C01815=1063.991,309.897,-98.913,173.800,33.597,156.214
C01816=1063.997,310.145,-98.945,173.803,33.601,156.215
C01817=1064.004,310.393,-98.978,173.806,33.605,156.216
C01818=1064.011,310.640,-99.011,173.809,33.609,156.217
C01819=1064.017,310.888,-99.044,173.812,33.614,156.218
C01820=1064.023,311.136,-99.077,173.815,33.618,156.219
C01821=1064.029,311.383,-99.109,173.818,33.622,156.220
C01822=1064.036,311.631,-99.142,173.821,33.626,156.220
C01823=1064.042,311.880,-99.175,173.824,33.631,156.221
C01824=1064.049,312.127,-99.207,173.828,33.635,156.222
C01825=1064.056,312.375,-99.239,173.832,33.640,156.223
C01826=1064.062,312.622,-99.272,173.835,33.644,156.224
C01827=1064.068,312.870,-99.305,173.838,33.648,156.225
C01828=1064.075,313.118,-99.338,173.841,33.652,156.225
C01829=1064.081,313.366,-99.371,173.844,33.657,156.226
C01830=1064.088,313.613,-99.404,173.847,33.661,156.227
C01831=1064.094,313.861,-99.436,173.850,33.665,156.228
C01832=1064.101,314.109,-99.469,173.853,33.670,156.229
C01833=1064.107,314.356,-99.503,173.858,33.674,156.230
C01834=1064.113,314.604,-99.536,173.861,33.679,156.231
C01835=1064.119,314.852,-99.570,173.864,33.683,156.232
C01836=1064.125,315.100,-99.602,173.867,33.688,156.233
C01837=1064.131,315.347,-99.635,173.870,33.692,156.233
C01838=1064.138,315.595,-99.669,173.873,33.697,156.234
C01839=1064.144,315.843,-99.702,173.876,33.701,156.235
C01840=1064.149,316.091,-99.736,173.879,33.705,156.236
C01841=1064.156,316.338,-99.768,173.883,33.710,156.237
C01842=1064.162,316.586,-99.802,173.887,33.714,156.238
C01843=1064.168,316.833,-99.835,173.890,33.719,156.239
C01844=1064.174,317.082,-99.869,173.893,33.723,156.240
C01845=1064.181,317.319,-99.901,173.896,33.728,156.241
C01846=1064.187,317.558,-99.933,173.899,33.732,156.242
C01847=1064.193,317.796,-99.965,173.902,33.736,156.242
C01848=1064.199,318.035,-99.997,173.905,33.741,156.243
C01849=1064.204,318.273,-100.029,173.909,33.745,156.244
C01850=1064.211,318.511,-100.061,173.912,33.749,156.245
C01851=1064.216,318.750,-100.093,173.915,33.754,156.246
C01852=1064.223,318.989,-100.126,173.918,33.758,156.247
C01853=1064.229,319.236,-100.160,173.921,33.762,156.248
C01854=1064.235,319.484,-100.192,173.925,33.767,156.249
C01855=1064.241,319.731,-100.227,173.928,33.772,156.249
C01856=1064.248,319.980,-100.260,173.931,33.776,156.250
C01857=1064.254,320.227,-100.294,173.935,33.781,156.251
C01858=1064.261,320.475,-100.327,173.938,33.785,156.252
C01859=1064.266,320.722,-100.361,173.941,33.789,156.253
C01860=1064.273,320.969,-100.394,173.945,33.794,156.254
C01861=1064.279,321.218,-100.428,173.948,33.799,156.255
C01862=1064.286,321.465,-100.461,173.951,33.803,156.256
C01863=1064.291,321.713,-100.495,173.954,33.808,156.257
C01864=1064.298,321.961,-100.529,173.959,33.813,156.258
C01865=1064.304,322.208,-100.563,173.962,33.817,156.259
C01866=1064.311,322.456,-100.596,173.965,33.821,156.260
C01867=1064.317,322.703,-100.630,173.968,33.826,156.260
C01868=1064.324,322.951,-100.664,173.971,33.831,156.261
C01869=1064.330,323.198,-100.698,173.975,33.835,156.262
C01870=1064.336,323.447,-100.731,173.979,33.840,156.263
C01871=1064.343,323.694,-100.765,173.982,33.844,156.264
C01872=1064.349,323.941,-100.799,173.985,33.849,156.265
C01873=1064.355,324.189,-100.833,173.989,33.853,156.266
C01874=1064.362,324.437,-100.866,173.992,33.858,156.267
C01875=1064.368,324.685,-100.901,173.995,33.863,156.268
C01876=1064.375,324.932,-100.934,173.998,33.867,156.269
C01877=1064.381,325.180,-100.968,174.003,33.872,156.270
C01878=1064.388,325.427,-101.002,174.006,33.876,156.271
C01879=1064.394,325.675,-101.036,174.009,33.881,156.272
C01880=1064.401,325.923,-101.071,174.012,33.886,156.273
C01881=1064.407,326.170,-101.104,174.016,33.890,156.273
C01882=1064.413,326.418,-101.138,174.019,33.895,156.274
C01883=1064.421,326.666,-101.172,174.023,33.899,156.275
C01884=1064.426,326.913,-101.206,174.027,33.904,156.276
C01885=1064.433,327.161,-101.240,174.030,33.909,156.277
C01886=1064.439,327.408,-101.274,174.033,33.913,156.278
C01887=1064.446,327.656,-101.308,174.036,33.918,156.279
C01888=1064.453,327.904,-101.343,174.040,33.923,156.280
C01889=1064.459,328.150,-101.377,174.044,33.928,156.281
C01890=1064.466,328.398,-101.411,174.047,33.932,156.282
C01891=1064.473,328.646,-101.445,174.051,33.936,156.283
C01892=1064.479,328.893,-101.479,174.054,33.941,156.284
C01893=1064.485,329.141,-101.513,174.057,33.946,156.285
C01894=1064.493,329.389,-101.547,174.061,33.950,156.286
C01895=1064.498,329.636,-101.581,174.065,33.955,156.287
C01896=1064.505,329.884,-101.616,174.068,33.960,156.288
C01897=1064.512,330.131,-101.650,174.072,33.965,156.289
C01898=1064.519,330.379,-101.685,174.075,33.969,156.290
C01899=1064.525,330.627,-101.719,174.078,33.974,156.291
C01900=1064.531,330.875,-101.753,174.083,33.979,156.291
C01901=1064.538,331.110,-101.786,174.086,33.983,156.292
C01902=1064.543,331.346,-101.819,174.089,33.987,156.293
C01903=1064.550,331.581,-101.852,174.092,33.992,156.294
C01904=1064.557,331.817,-101.885,174.096,33.997,156.295
C01905=1064.562,332.052,-101.918,174.099,34.002,156.296
C01906=1064.568,332.287,-101.950,174.103,34.006,156.297
C01907=1064.574,332.523,-101.984,174.106,34.010,156.298
C01908=1064.580,332.759,-102.016,174.109,34.015,156.299
C01909=1064.587,333.006,-102.051,174.113,34.020,156.300
C01910=1064.593,333.254,-102.085,174.116,34.025,156.301
C01911=1064.600,333.501,-102.120,174.120,34.030,156.302
C01912=1064.606,333.749,-102.155,174.124,34.034,156.303
C01913=1064.613,333.996,-102.190,174.127,34.040,156.304
C01914=1064.619,334.244,-102.224,174.131,34.044,156.305
C01915=1064.626,334.491,-102.259,174.134,34.049,156.306
C01916=1064.631,334.739,-102.294,174.138,34.054,156.307
C01917=1064.638,334.987,-102.329,174.142,34.059,156.308
C01918=1064.645,335.234,-102.364,174.145,34.064,156.309
C01919=1064.651,335.482,-102.399,174.149,34.068,156.310
C01920=1064.657,335.729,-102.434,174.152,34.073,156.311
C01921=1064.664,335.977,-102.468,174.156,34.078,156.312
C01922=1064.671,336.224,-102.503,174.160,34.083,156.313
C01923=1064.677,336.471,-102.538,174.163,34.088,156.314
C01924=1064.684,336.719,-102.573,174.167,34.093,156.315
C01925=1064.691,336.967,-102.608,174.170,34.098,156.316
C01926=1064.697,337.214,-102.643,174.174,34.103,156.317
C01927=1064.704,337.462,-102.679,174.178,34.107,156.318
C01928=1064.710,337.708,-102.714,174.181,34.113,156.319
C01929=1064.716,337.956,-102.749,174.185,34.118,156.320
C01930=1064.723,338.204,-102.783,174.189,34.122,156.321
C01931=1064.729,338.451,-102.819,174.193,34.128,156.322
C01932=1064.736,338.699,-102.854,174.196,34.132,156.323
C01933=1064.742,338.946,-102.889,174.200,34.138,156.324
C01934=1064.748,339.194,-102.925,174.203,34.142,156.325
C01935=1064.755,339.441,-102.960,174.207,34.147,156.326
C01936=1064.762,339.688,-102.995,174.211,34.153,156.327
C01937=1064.767,339.935,-103.030,174.214,34.157,156.328
C01938=1064.774,340.183,-103.066,174.218,34.163,156.330
C01939=1064.781,340.430,-103.101,174.222,34.168,156.331
C01940=1064.788,340.678,-103.136,174.226,34.172,156.332
C01941=1064.794,340.925,-103.172,174.229,34.178,156.333
C01942=1064.801,341.173,-103.207,174.233,34.183,156.334
C01943=1064.807,341.420,-103.242,174.237,34.188,156.335
C01944=1064.813,341.668,-103.278,174.241,34.193,156.336
C01945=1064.820,341.915,-103.313,174.244,34.198,156.337
C01946=1064.826,342.162,-103.349,174.248,34.203,156.338
C01947=1064.833,342.409,-103.384,174.252,34.208,156.339
C01948=1064.840,342.657,-103.419,174.256,34.213,156.340
C01949=1064.847,342.905,-103.456,174.259,34.218,156.341
C01950=1064.853,343.153,-103.491,174.263,34.223,156.342
C01951=1064.860,343.399,-103.527,174.267,34.228,156.343
C01952=1064.867,343.647,-103.562,174.271,34.233,156.344
C01953=1064.873,343.894,-103.597,174.274,34.239,156.345
C01954=1064.879,344.142,-103.633,174.278,34.244,156.347
C01955=1064.886,344.389,-103.669,174.282,34.249,156.348
C01956=1064.892,344.636,-103.705,174.286,34.254,156.349
C01957=1064.899,344.869,-103.739,174.289,34.259,156.350
C01958=1064.905,345.102,-103.772,174.293,34.264,156.351
C01959=1064.911,345.336,-103.806,174.297,34.269,156.352
C01960=1064.917,345.569,-103.839,174.300,34.274,156.353
C01961=1064.923,345.802,-103.874,174.304,34.279,156.354
C01962=1064.929,346.035,-103.908,174.307,34.284,156.355
C01963=1064.936,346.268,-103.942,174.311,34.288,156.356
C01964=1064.942,346.501,-103.975,174.315,34.294,156.357
C01965=1064.948,346.748,-104.011,174.318,34.299,156.358
C01966=1064.955,346.997,-104.047,174.322,34.304,156.359
C01967=1064.962,347.244,-104.083,174.327,34.309,156.360
C01968=1064.968,347.491,-104.119,174.330,34.314,156.361
C01969=1064.975,347.738,-104.155,174.334,34.320,156.363
C01970=1064.981,347.985,-104.191,174.338,34.325,156.364
C01971=1064.988,348.232,-104.227,174.342,34.331,156.365
C01972=1064.995,348.480,-104.263,174.346,34.336,156.366
C01973=1065.001,348.727,-104.299,174.349,34.341,156.367
C01974=1065.008,348.974,-104.336,174.354,34.346,156.368
C01975=1065.014,349.222,-104.371,174.357,34.351,156.369
C01976=1065.021,349.469,-104.408,174.361,34.357,156.370
C01977=1065.028,349.717,-104.444,174.366,34.362,156.372
C01978=1065.034,349.964,-104.481,174.369,34.367,156.373
C01979=1065.041,350.211,-104.516,174.373,34.373,156.374
C01980=1065.048,350.459,-104.553,174.376,34.378,156.375
C01981=1065.054,350.706,-104.589,174.381,34.384,156.376
C01982=1065.061,350.952,-104.625,174.385,34.389,156.377
C01983=1065.068,351.200,-104.662,174.388,34.394,156.378
C01984=1065.074,351.447,-104.698,174.393,34.400,156.380
C01985=1065.081,351.694,-104.735,174.397,34.405,156.381
C01986=1065.088,351.942,-104.771,174.400,34.411,156.382
C01987=1065.095,352.189,-104.807,174.405,34.416,156.383
C01988=1065.101,352.436,-104.844,174.409,34.422,156.384
C01989=1065.107,352.683,-104.880,174.412,34.427,156.385
C01990=1065.114,352.931,-104.917,174.417,34.432,156.387
C01991=1065.121,353.178,-104.953,174.421,34.438,156.388
C01992=1065.128,353.426,-104.990,174.424,34.443,156.389
C01993=1065.134,353.673,-105.027,174.428,34.449,156.390
C01994=1065.140,353.920,-105.063,174.433,34.454,156.391
C01995=1065.147,354.167,-105.100,174.436,34.460,156.392
C01996=1065.154,354.414,-105.137,174.440,34.466,156.394
C01997=1065.160,354.661,-105.174,174.445,34.471,156.395
C01998=1065.167,354.909,-105.210,174.449,34.477,156.396
C01999=1065.173,355.156,-105.247,174.452,34.482,156.397
C02000=1065.180,355.403,-105.284,174.457,34.488,156.398
C02001=1065.187,355.650,-105.321,174.461,34.493,156.400
C02002=1065.194,355.898,-105.358,174.464,34.499,156.401
C02003=1065.200,356.145,-105.394,174.469,34.505,156.402
C02004=1065.207,356.391,-105.431,174.473,34.510,156.403
C02005=1065.214,356.639,-105.468,174.477,34.516,156.404
C02006=1065.220,356.886,-105.504,174.481,34.521,156.406
C02007=1065.227,357.133,-105.542,174.485,34.527,156.407
C02008=1065.234,357.380,-105.578,174.490,34.533,156.408
C02009=1065.241,357.627,-105.616,174.494,34.538,156.409
C02010=1065.248,357.875,-105.653,174.497,34.544,156.410
C02011=1065.255,358.121,-105.690,174.502,34.549,156.412
C02012=1065.262,358.369,-105.727,174.506,34.555,156.413
C02013=1065.268,358.604,-105.762,174.509,34.561,156.414
C02014=1065.274,358.839,-105.798,174.514,34.566,156.415
C02015=1065.280,359.074,-105.833,174.518,34.572,156.416
C02016=1065.287,359.309,-105.868,174.521,34.577,156.418
C02017=1065.293,359.544,-105.904,174.526,34.582,156.419
C02018=1065.300,359.780,-105.939,174.529,34.588,156.420
C02019=1065.306,360.015,-105.974,174.533,34.593,156.421
C02020=1065.312,360.250,-106.010,174.538,34.599,156.422
C02021=1065.319,360.497,-106.048,174.541,34.605,156.424
C02022=1065.326,360.744,-106.085,174.546,34.610,156.425
C02023=1065.333,360.991,-106.122,174.550,34.616,156.426
C02024=1065.340,361.239,-106.160,174.554,34.622,156.427
C02025=1065.346,361.485,-106.197,174.559,34.628,156.429
C02026=1065.353,361.732,-106.234,174.563,34.634,156.430
C02027=1065.360,361.980,-106.271,174.566,34.639,156.431
C02028=1065.367,362.227,-106.308,174.571,34.645,156.432
C02029=1065.374,362.474,-106.347,174.575,34.651,156.434
C02030=1065.381,362.721,-106.384,174.580,34.657,156.435
C02031=1065.387,362.968,-106.421,174.584,34.663,156.436
C02032=1065.394,363.215,-106.459,174.588,34.669,156.438
C02033=1065.401,363.462,-106.497,174.592,34.675,156.439
C02034=1065.408,363.709,-106.534,174.596,34.680,156.440
C02035=1065.414,363.956,-106.572,174.601,34.687,156.442
C02036=1065.422,364.203,-106.610,174.605,34.692,156.443
C02037=1065.429,364.450,-106.647,174.609,34.698,156.444
C02038=1065.435,364.697,-106.685,174.614,34.704,156.445
C02039=1065.442,364.944,-106.722,174.618,34.710,156.447
C02040=1065.448,365.192,-106.761,174.623,34.717,156.448
C02041=1065.455,365.438,-106.798,174.626,34.722,156.449
C02042=1065.462,365.685,-106.837,174.631,34.728,156.451
C02043=1065.468,365.932,-106.875,174.635,34.735,156.452
C02044=1065.476,366.180,-106.912,174.639,34.740,156.453
C02045=1065.482,366.426,-106.951,174.644,34.747,156.455
C02046=1065.489,366.673,-106.988,174.648,34.753,156.456
C02047=1065.496,366.920,-107.026,174.653,34.759,156.457
C02048=1065.503,367.167,-107.065,174.657,34.765,156.459
C02049=1065.510,367.414,-107.103,174.662,34.771,156.460
C02050=1065.517,367.661,-107.140,174.666,34.777,156.461
C02051=1065.523,367.907,-107.179,174.669,34.783,156.463
C02052=1065.530,368.155,-107.217,174.674,34.790,156.464
C02053=1065.537,368.401,-107.255,174.678,34.796,156.466
C02054=1065.544,368.649,-107.293,174.683,34.802,156.467
C02055=1065.551,368.896,-107.331,174.687,34.808,156.468
C02056=1065.558,369.143,-107.370,174.692,34.814,156.470
C02057=1065.565,369.390,-107.408,174.696,34.820,156.471
C02058=1065.572,369.637,-107.446,174.701,34.826,156.472
C02059=1065.579,369.884,-107.485,174.705,34.832,156.474
C02060=1065.585,370.130,-107.522,174.710,34.839,156.475
C02061=1065.592,370.377,-107.561,174.714,34.845,156.477
C02062=1065.599,370.624,-107.600,174.719,34.852,156.478
C02063=1065.606,370.871,-107.637,174.723,34.858,156.479
C02064=1065.613,371.118,-107.676,174.728,34.864,156.481
C02065=1065.620,371.365,-107.715,174.732,34.870,156.482
C02066=1065.627,371.612,-107.752,174.736,34.876,156.483
C02067=1065.634,371.858,-107.791,174.741,34.883,156.485
C02068=1065.641,372.105,-107.830,174.745,34.889,156.486
C02069=1065.648,372.349,-107.868,174.750,34.896,156.488
C02070=1065.655,372.594,-107.906,174.754,34.902,156.489
C02071=1065.662,372.837,-107.944,174.759,34.908,156.490
C02072=1065.668,373.081,-107.982,174.763,34.914,156.492
C02073=1065.675,373.325,-108.021,174.768,34.921,156.493
C02074=1065.683,373.569,-108.059,174.772,34.927,156.495
C02075=1065.689,373.812,-108.097,174.777,34.933,156.496
C02076=1065.696,374.057,-108.135,174.781,34.940,156.498
C02077=1065.703,374.304,-108.174,174.786,34.946,156.499
C02078=1065.709,374.550,-108.213,174.790,34.953,156.501
C02079=1065.716,374.797,-108.252,174.795,34.960,156.502
C02080=1065.723,375.044,-108.291,174.800,34.966,156.503
C02081=1065.730,375.291,-108.330,174.804,34.972,156.505
C02082=1065.738,375.538,-108.370,174.809,34.979,156.506
C02083=1065.744,375.785,-108.408,174.813,34.985,156.508
C02084=1065.751,376.031,-108.447,174.818,34.992,156.509
C02085=1065.758,376.278,-108.486,174.823,34.999,156.511
C02086=1065.766,376.525,-108.524,174.828,35.006,156.512
C02087=1065.773,376.771,-108.564,174.832,35.012,156.514
C02088=1065.780,377.018,-108.603,174.837,35.018,156.515
C02089=1065.787,377.265,-108.642,174.841,35.025,156.517
C02090=1065.794,377.511,-108.681,174.846,35.032,156.518
C02091=1065.801,377.758,-108.720,174.851,35.039,156.520
C02092=1065.808,378.005,-108.759,174.855,35.045,156.521
C02093=1065.815,378.252,-108.799,174.861,35.052,156.523
C02094=1065.822,378.499,-108.838,174.865,35.059,156.524
C02095=1065.829,378.745,-108.877,174.870,35.065,156.526
C02096=1065.836,378.992,-108.916,174.874,35.072,156.527
C02097=1065.843,379.239,-108.957,174.879,35.079,156.529
C02098=1065.850,379.486,-108.996,174.884,35.085,156.530
C02099=1065.857,379.732,-109.035,174.889,35.092,156.532
C02100=1065.864,379.980,-109.074,174.894,35.099,156.533
C02101=1065.872,380.226,-109.114,174.898,35.106,156.535
C02102=1065.878,380.473,-109.153,174.903,35.113,156.537
C02103=1065.886,380.720,-109.193,174.907,35.119,156.538
C02104=1065.893,380.966,-109.232,174.912,35.126,156.540
C02105=1065.900,381.213,-109.271,174.918,35.133,156.541
C02106=1065.908,381.460,-109.311,174.922,35.140,156.543
C02107=1065.914,381.706,-109.351,174.927,35.147,156.544
C02108=1065.921,381.952,-109.391,174.932,35.154,156.546
C02109=1065.929,382.199,-109.431,174.936,35.161,156.548
C02110=1065.935,382.446,-109.470,174.942,35.168,156.549
C02111=1065.943,382.693,-109.510,174.946,35.175,156.551
C02112=1065.950,382.939,-109.550,174.951,35.182,156.552
C02113=1065.956,383.186,-109.590,174.956,35.189,156.554
C02114=1065.964,383.433,-109.630,174.961,35.196,156.556
C02115=1065.971,383.679,-109.669,174.966,35.203,156.557
C02116=1065.978,383.926,-109.710,174.971,35.210,156.559
C02117=1065.985,384.172,-109.749,174.975,35.217,156.560
C02118=1065.992,384.419,-109.789,174.981,35.224,156.562
C02119=1065.999,384.666,-109.829,174.986,35.232,156.564
C02120=1066.006,384.912,-109.869,174.990,35.238,156.565
C02121=1066.014,385.159,-109.910,174.996,35.246,156.567
C02122=1066.021,385.405,-109.950,175.001,35.253,156.569
C02123=1066.029,385.652,-109.990,175.005,35.260,156.570
C02124=1066.036,385.899,-110.030,175.010,35.267,156.572
C02125=1066.044,386.170,-110.074,175.016,35.275,156.574
C02126=1066.052,386.441,-110.119,175.021,35.283,156.576
C02127=1066.060,386.712,-110.163,175.027,35.291,156.577
C02128=1066.067,386.984,-110.206,175.032,35.299,156.579
C02129=1066.075,387.231,-110.248,175.038,35.306,156.581
C02130=1066.082,387.477,-110.287,175.042,35.314,156.583
C02131=1066.090,387.723,-110.328,175.048,35.321,156.584
C02132=1066.097,387.970,-110.368,175.053,35.328,156.586
C02133=1066.104,388.217,-110.408,175.057,35.336,156.588
C02134=1066.111,388.463,-110.449,175.063,35.343,156.589
C02135=1066.119,388.710,-110.489,175.068,35.350,156.591
C02136=1066.126,388.956,-110.530,175.073,35.358,156.593
C02137=1066.133,389.203,-110.570,175.078,35.365,156.595
C02138=1066.141,389.449,-110.611,175.083,35.372,156.596
C02139=1066.148,389.695,-110.651,175.089,35.380,156.598
C02140=1066.155,389.942,-110.692,175.094,35.387,156.600
C02141=1066.163,390.189,-110.732,175.098,35.395,156.601
C02142=1066.170,390.435,-110.774,175.104,35.402,156.603
C02143=1066.178,390.682,-110.814,175.109,35.410,156.605
C02144=1066.185,390.928,-110.854,175.115,35.417,156.607
C02145=1066.192,391.175,-110.896,175.119,35.425,156.608
C02146=1066.200,391.421,-110.936,175.125,35.432,156.610
C02147=1066.207,391.668,-110.977,175.130,35.440,156.612
C02148=1066.214,391.914,-111.018,175.136,35.448,156.614
C02149=1066.222,392.160,-111.058,175.140,35.455,156.616
C02150=1066.229,392.407,-111.099,175.146,35.463,156.617
C02151=1066.236,392.653,-111.141,175.151,35.471,156.619
C02152=1066.244,392.900,-111.182,175.156,35.478,156.621
C02153=1066.252,393.146,-111.223,175.162,35.486,156.623
C02154=1066.258,393.392,-111.263,175.166,35.494,156.625
C02155=1066.266,393.639,-111.305,175.172,35.501,156.626
C02156=1066.273,393.885,-111.346,175.177,35.509,156.628
C02157=1066.280,394.132,-111.387,175.183,35.517,156.630
C02158=1066.288,394.378,-111.428,175.188,35.525,156.632
C02159=1066.296,394.624,-111.470,175.193,35.533,156.634
C02160=1066.303,394.871,-111.511,175.199,35.541,156.636
C02161=1066.310,395.117,-111.552,175.204,35.548,156.637
C02162=1066.318,395.364,-111.593,175.210,35.556,156.639
C02163=1066.325,395.610,-111.635,175.215,35.564,156.641
C02164=1066.332,395.857,-111.677,175.221,35.572,156.643
C02165=1066.340,396.103,-111.718,175.226,35.580,156.645
C02166=1066.347,396.349,-111.760,175.231,35.588,156.647
C02167=1066.355,396.596,-111.801,175.236,35.596,156.649
C02168=1066.362,396.842,-111.842,175.242,35.604,156.651
C02169=1066.370,397.088,-111.884,175.248,35.612,156.652
C02170=1066.377,397.335,-111.925,175.253,35.620,156.654
C02171=1066.385,397.581,-111.967,175.259,35.628,156.656
C02172=1066.392,397.827,-112.008,175.264,35.636,156.658
C02173=1066.400,398.074,-112.051,175.270,35.645,156.660
C02174=1066.407,398.321,-112.092,175.276,35.653,156.662
C02175=1066.415,398.567,-112.134,175.280,35.661,156.664
C02176=1066.422,398.813,-112.176,175.286,35.669,156.666
C02177=1066.430,399.059,-112.217,175.291,35.677,156.668
C02178=1066.437,399.305,-112.259,175.297,35.685,156.670
C02179=1066.445,399.551,-112.301,175.303,35.694,156.672
C02180=1066.452,399.798,-112.344,175.308,35.702,156.674
C02181=1066.462,400.119,-112.398,175.315,35.713,156.676
C02182=1066.472,400.440,-112.453,175.324,35.724,156.679
C02183=1066.482,400.761,-112.507,175.331,35.734,156.681
C02184=1066.492,401.081,-112.562,175.338,35.745,156.684
C02185=1066.499,401.327,-112.604,175.343,35.754,156.686
C02186=1066.507,401.574,-112.647,175.349,35.762,156.688
C02187=1066.515,401.820,-112.689,175.355,35.771,156.690
C02188=1066.522,402.067,-112.731,175.361,35.779,156.692
C02189=1066.530,402.313,-112.773,175.366,35.788,156.694
C02190=1066.538,402.559,-112.815,175.372,35.796,156.696
C02191=1066.546,402.806,-112.858,175.378,35.804,156.698
C02192=1066.553,403.052,-112.900,175.384,35.813,156.700
C02193=1066.560,403.298,-112.942,175.389,35.822,156.702
C02194=1066.569,403.544,-112.985,175.395,35.830,156.705
C02195=1066.576,403.790,-113.028,175.401,35.839,156.707
C02196=1066.584,404.037,-113.070,175.407,35.848,156.709
C02197=1066.591,404.283,-113.113,175.413,35.856,156.711
C02198=1066.599,404.529,-113.156,175.418,35.865,156.713
C02199=1066.607,404.775,-113.197,175.424,35.874,156.715
C02200=1066.615,405.022,-113.241,175.430,35.882,156.717
C02201=1066.622,405.268,-113.283,175.436,35.891,156.719
C02202=1066.630,405.515,-113.326,175.442,35.900,156.721
C02203=1066.638,405.760,-113.369,175.449,35.909,156.723
C02204=1066.645,406.007,-113.412,175.454,35.917,156.726
C02205=1066.652,406.236,-113.452,175.460,35.926,156.728
C02206=1066.660,406.466,-113.492,175.465,35.934,156.730
C02207=1066.667,406.695,-113.532,175.471,35.942,156.732
C02208=1066.674,406.924,-113.572,175.477,35.951,156.734
C02209=1066.681,407.155,-113.612,175.482,35.959,156.736
C02210=1066.688,407.384,-113.652,175.488,35.968,156.738
C02211=1066.696,407.614,-113.692,175.493,35.976,156.740
C02212=1066.703,407.843,-113.732,175.499,35.984,156.742
C02213=1066.710,408.090,-113.776,175.505,35.993,156.744
C02214=1066.718,408.335,-113.819,175.511,36.003,156.746
C02215=1066.726,408.581,-113.862,175.517,36.012,156.748
C02216=1066.733,408.828,-113.905,175.524,36.021,156.751
C02217=1066.741,409.074,-113.948,175.530,36.030,156.753
C02218=1066.749,409.320,-113.991,175.536,36.039,156.755
C02219=1066.757,409.566,-114.035,175.542,36.048,156.757
C02220=1066.765,409.812,-114.078,175.548,36.057,156.760
C02221=1066.773,410.058,-114.121,175.555,36.067,156.762
C02222=1066.780,410.304,-114.165,175.561,36.076,156.764
C02223=1066.788,410.551,-114.209,175.567,36.085,156.766
C02224=1066.797,410.796,-114.252,175.573,36.095,156.769
C02225=1066.805,411.043,-114.296,175.579,36.104,156.771
C02226=1066.812,411.289,-114.340,175.586,36.113,156.773
C02227=1066.820,411.534,-114.382,175.592,36.123,156.776
C02228=1066.828,411.781,-114.426,175.598,36.133,156.778
C02229=1066.836,412.026,-114.470,175.604,36.142,156.780
C02230=1066.844,412.273,-114.514,175.611,36.151,156.783
C02231=1066.852,412.519,-114.557,175.617,36.161,156.785
C02232=1066.860,412.765,-114.601,175.623,36.170,156.787
C02233=1066.868,413.011,-114.645,175.631,36.180,156.790
C02234=1066.876,413.257,-114.689,175.637,36.189,156.792
C02235=1066.884,413.503,-114.733,175.643,36.199,156.794
C02236=1066.893,413.748,-114.776,175.649,36.209,156.797
C02237=1066.903,414.041,-114.829,175.657,36.220,156.800
C02238=1066.912,414.333,-114.881,175.665,36.231,156.802
C02239=1066.921,414.625,-114.933,175.673,36.243,156.805
C02240=1066.931,414.917,-114.985,175.681,36.254,156.808
C02241=1066.939,415.163,-115.030,175.687,36.265,156.811
C02242=1066.947,415.408,-115.074,175.693,36.274,156.813
C02243=1066.955,415.655,-115.118,175.701,36.284,156.816
C02244=1066.963,415.900,-115.162,175.707,36.294,156.818
C02245=1066.971,416.146,-115.206,175.714,36.304,156.821
C02246=1066.979,416.393,-115.252,175.720,36.314,156.823
C02247=1066.987,416.639,-115.296,175.728,36.324,156.826
C02248=1066.995,416.884,-115.340,175.734,36.334,156.828
C02249=1067.003,417.130,-115.385,175.740,36.344,156.830
C02250=1067.011,417.376,-115.429,175.748,36.354,156.833
C02251=1067.019,417.622,-115.473,175.754,36.364,156.836
C02252=1067.028,417.868,-115.518,175.761,36.374,156.838
C02253=1067.036,418.114,-115.562,175.768,36.384,156.841
C02254=1067.044,418.359,-115.607,175.775,36.394,156.843
C02255=1067.052,418.605,-115.652,175.781,36.405,156.846
C02256=1067.060,418.851,-115.697,175.789,36.415,156.848
C02257=1067.068,419.097,-115.741,175.795,36.425,156.851
C02258=1067.077,419.342,-115.786,175.803,36.436,156.854
C02259=1067.085,419.589,-115.831,175.809,36.446,156.856
C02260=1067.094,419.835,-115.875,175.816,36.456,156.859
C02261=1067.102,420.081,-115.921,175.823,36.466,156.861
C02262=1067.110,420.326,-115.966,175.830,36.477,156.864
C02263=1067.118,420.572,-116.011,175.837,36.488,156.867
C02264=1067.127,420.818,-116.056,175.844,36.498,156.869
C02265=1067.135,421.063,-116.101,175.851,36.508,156.872
C02266=1067.144,421.309,-116.147,175.858,36.519,156.874
C02267=1067.152,421.555,-116.191,175.866,36.529,156.877
C02268=1067.159,421.800,-116.237,175.872,36.540,156.880
C02269=1067.168,422.046,-116.282,175.880,36.551,156.883
C02270=1067.176,422.292,-116.328,175.887,36.562,156.885
C02271=1067.185,422.538,-116.372,175.894,36.572,156.888
C02272=1067.193,422.783,-116.417,175.902,36.583,156.891
C02273=1067.201,423.029,-116.463,175.909,36.594,156.894
C02274=1067.210,423.275,-116.509,175.916,36.605,156.896
C02275=1067.218,423.521,-116.554,175.923,36.615,156.899
C02276=1067.227,423.766,-116.600,175.931,36.626,156.902
C02277=1067.234,424.012,-116.646,175.938,36.637,156.905
C02278=1067.243,424.258,-116.691,175.945,36.648,156.907
C02279=1067.252,424.504,-116.737,175.953,36.659,156.910
C02280=1067.260,424.748,-116.783,175.960,36.670,156.913
C02281=1067.269,424.994,-116.829,175.967,36.681,156.916
C02282=1067.277,425.240,-116.874,175.975,36.692,156.919
C02283=1067.285,425.486,-116.920,175.983,36.703,156.921
C02284=1067.294,425.731,-116.966,175.990,36.714,156.924
C02285=1067.303,425.977,-117.012,175.997,36.726,156.927
C02286=1067.312,426.223,-117.057,176.005,36.737,156.930
C02287=1067.320,426.468,-117.104,176.013,36.748,156.933
C02288=1067.329,426.714,-117.149,176.021,36.759,156.936
C02289=1067.337,426.959,-117.196,176.028,36.770,156.939
C02290=1067.346,427.205,-117.241,176.035,36.782,156.942
C02291=1067.355,427.450,-117.288,176.043,36.793,156.945
C02292=1067.363,427.696,-117.335,176.051,36.804,156.948
C02293=1067.374,428.007,-117.393,176.061,36.819,156.951
C02294=1067.385,428.318,-117.452,176.071,36.833,156.955
C02295=1067.396,428.630,-117.511,176.080,36.848,156.959
C02296=1067.407,428.942,-117.570,176.091,36.863,156.963
C02297=1067.415,429.186,-117.616,176.099,36.874,156.966
C02298=1067.423,429.432,-117.663,176.106,36.886,156.969
C02299=1067.433,429.677,-117.709,176.114,36.898,156.972
C02300=1067.441,429.923,-117.756,176.122,36.910,156.975
C02301=1067.450,430.168,-117.803,176.130,36.921,156.978
C02302=1067.458,430.414,-117.849,176.138,36.933,156.981
C02303=1067.468,430.660,-117.896,176.146,36.945,156.984
C02304=1067.477,430.905,-117.943,176.154,36.957,156.987
C02305=1067.485,431.151,-117.989,176.162,36.969,156.990
C02306=1067.494,431.396,-118.036,176.170,36.980,156.993
C02307=1067.503,431.641,-118.084,176.178,36.992,156.997
C02308=1067.511,431.887,-118.130,176.186,37.004,157.000
C02309=1067.520,432.131,-118.178,176.195,37.017,157.003
C02310=1067.528,432.377,-118.224,176.203,37.029,157.006
C02311=1067.537,432.622,-118.272,176.211,37.041,157.009
C02312=1067.546,432.868,-118.319,176.220,37.053,157.012
C02313=1067.555,433.113,-118.366,176.228,37.066,157.016
C02314=1067.564,433.358,-118.413,176.236,37.078,157.019
C02315=1067.572,433.604,-118.461,176.244,37.090,157.022
C02316=1067.581,433.849,-118.509,176.252,37.102,157.025
C02317=1067.590,434.094,-118.556,176.262,37.115,157.029
C02318=1067.599,434.340,-118.603,176.270,37.127,157.032
C02319=1067.608,434.585,-118.651,176.278,37.140,157.035
C02320=1067.617,434.830,-118.698,176.286,37.152,157.039
C02321=1067.626,435.075,-118.746,176.296,37.164,157.042
C02322=1067.635,435.321,-118.794,176.304,37.177,157.045
C02323=1067.644,435.565,-118.841,176.312,37.190,157.049
C02324=1067.653,435.810,-118.889,176.321,37.202,157.052
C02325=1067.662,436.056,-118.937,176.330,37.215,157.055
C02326=1067.671,436.301,-118.984,176.338,37.227,157.059
C02327=1067.680,436.547,-119.032,176.348,37.240,157.062
C02328=1067.689,436.791,-119.080,176.356,37.253,157.066
C02329=1067.699,437.037,-119.128,176.364,37.266,157.069
C02330=1067.708,437.282,-119.176,176.374,37.279,157.072
C02331=1067.717,437.527,-119.224,176.382,37.292,157.076
C02332=1067.726,437.772,-119.273,176.392,37.305,157.079
C02333=1067.735,438.017,-119.320,176.400,37.318,157.083
C02334=1067.745,438.262,-119.369,176.409,37.331,157.086
C02335=1067.754,438.508,-119.416,176.418,37.344,157.090
C02336=1067.763,438.752,-119.465,176.427,37.357,157.093
C02337=1067.772,438.997,-119.514,176.436,37.370,157.097
C02338=1067.782,439.243,-119.561,176.446,37.383,157.100
C02339=1067.790,439.488,-119.610,176.454,37.397,157.104
C02340=1067.800,439.733,-119.659,176.464,37.410,157.108
C02341=1067.809,439.978,-119.708,176.472,37.423,157.111
C02342=1067.819,440.223,-119.756,176.482,37.437,157.115
C02343=1067.828,440.467,-119.805,176.491,37.450,157.119
C02344=1067.837,440.712,-119.854,176.500,37.464,157.122
C02345=1067.847,440.957,-119.902,176.510,37.477,157.126
C02346=1067.856,441.203,-119.951,176.519,37.491,157.130
C02347=1067.866,441.448,-120.000,176.528,37.505,157.133
C02348=1067.875,441.693,-120.049,176.538,37.518,157.137
C02349=1067.886,442.009,-120.113,176.550,37.536,157.142
C02350=1067.899,442.325,-120.175,176.562,37.554,157.147
C02351=1067.910,442.641,-120.239,176.575,37.571,157.152
C02352=1067.923,442.957,-120.302,176.588,37.590,157.157
C02353=1067.932,443.202,-120.352,176.596,37.604,157.160
C02354=1067.942,443.447,-120.401,176.606,37.618,157.164
C02355=1067.951,443.692,-120.450,176.616,37.631,157.168
C02356=1067.961,443.937,-120.500,176.626,37.646,157.172
C02357=1067.970,444.182,-120.548,176.636,37.660,157.176
C02358=1067.980,444.427,-120.598,176.646,37.674,157.180
C02359=1067.990,444.672,-120.648,176.656,37.688,157.184
C02360=1067.999,444.916,-120.698,176.666,37.703,157.188
C02361=1068.009,445.161,-120.747,176.676,37.717,157.191
C02362=1068.018,445.405,-120.797,176.686,37.731,157.196
C02363=1068.028,445.650,-120.847,176.696,37.746,157.199
C02364=1068.038,445.895,-120.897,176.706,37.760,157.204
C02365=1068.048,446.140,-120.947,176.716,37.775,157.208
C02366=1068.057,446.384,-120.996,176.726,37.789,157.212
C02367=1068.067,446.630,-121.047,176.736,37.804,157.216
C02368=1068.076,446.874,-121.096,176.746,37.819,157.220
C02369=1068.087,447.118,-121.146,176.757,37.833,157.224
C02370=1068.097,447.364,-121.197,176.767,37.848,157.228
C02371=1068.106,447.608,-121.246,176.778,37.863,157.232
C02372=1068.116,447.853,-121.297,176.788,37.878,157.236
C02373=1068.126,448.096,-121.347,176.798,37.893,157.240
C02374=1068.137,448.339,-121.396,176.809,37.907,157.244
C02375=1068.149,448.584,-121.445,176.820,37.921,157.248
C02376=1068.162,448.829,-121.492,176.830,37.935,157.252
C02377=1068.177,449.073,-121.539,176.839,37.948,157.256
C02378=1068.193,449.319,-121.586,176.849,37.961,157.260
C02379=1068.209,449.564,-121.632,176.858,37.974,157.263
C02380=1068.227,449.809,-121.677,176.867,37.986,157.267
C02381=1067.882,449.811,-121.936,176.856,38.119,157.302
C02382=1067.864,449.566,-121.891,176.846,38.107,157.299
C02383=1067.848,449.321,-121.845,176.837,38.094,157.295
C02384=1067.832,449.076,-121.799,176.827,38.081,157.292
C02385=1067.818,448.831,-121.751,176.817,38.068,157.288
C02386=1067.805,448.586,-121.703,176.807,38.054,157.284
C02387=1067.792,448.341,-121.654,176.796,38.040,157.280
C02388=1067.780,448.098,-121.605,176.786,38.026,157.276
C02389=1067.770,447.855,-121.556,176.775,38.011,157.272
C02390=1067.760,447.610,-121.505,176.765,37.997,157.268
C02391=1067.751,447.366,-121.455,176.754,37.982,157.264
C02392=1067.741,447.120,-121.405,176.744,37.967,157.259
C02393=1067.730,446.877,-121.355,176.733,37.952,157.255
C02394=1067.721,446.632,-121.305,176.723,37.938,157.251
C02395=1067.711,446.387,-121.255,176.713,37.923,157.247
C02396=1067.702,446.142,-121.205,176.703,37.909,157.243
C02397=1067.691,445.898,-121.155,176.693,37.894,157.239
C02398=1067.682,445.653,-121.105,176.682,37.879,157.235
C02399=1067.672,445.408,-121.055,176.672,37.865,157.231
C02400=1067.663,445.164,-121.005,176.661,37.851,157.227
C02401=1067.653,444.919,-120.956,176.652,37.836,157.223
C02402=1067.643,444.674,-120.906,176.642,37.822,157.219
C02403=1067.634,444.429,-120.856,176.632,37.808,157.215
C02404=1067.625,444.184,-120.807,176.622,37.794,157.211
C02405=1067.614,443.940,-120.757,176.612,37.780,157.207
C02406=1067.605,443.695,-120.707,176.602,37.766,157.203
C02407=1067.596,443.450,-120.658,176.592,37.752,157.200
C02408=1067.585,443.205,-120.609,176.582,37.738,157.196
C02409=1067.576,442.960,-120.559,176.572,37.724,157.192
C02410=1067.565,442.662,-120.500,176.561,37.707,157.187
C02411=1067.553,442.366,-120.441,176.549,37.690,157.183
C02412=1067.541,442.068,-120.380,176.538,37.673,157.178
C02413=1067.530,441.771,-120.321,176.525,37.657,157.174
C02414=1067.520,441.526,-120.272,176.517,37.643,157.170
C02415=1067.511,441.281,-120.223,176.507,37.629,157.166
C02416=1067.503,441.037,-120.174,176.497,37.616,157.162
C02417=1067.493,440.792,-120.126,176.488,37.602,157.159
C02418=1067.484,440.546,-120.076,176.478,37.589,157.155
C02419=1067.474,440.301,-120.028,176.469,37.575,157.151
C02420=1067.464,440.056,-119.979,176.460,37.562,157.148
C02421=1067.455,439.811,-119.930,176.450,37.549,157.144
C02422=1067.446,439.567,-119.882,176.441,37.535,157.140
C02423=1067.437,439.321,-119.833,176.432,37.522,157.137
C02424=1067.428,439.077,-119.784,176.423,37.509,157.133
C02425=1067.418,438.831,-119.737,176.414,37.496,157.130
C02426=1067.410,438.586,-119.688,176.404,37.483,157.126
C02427=1067.400,438.341,-119.639,176.396,37.470,157.123
C02428=1067.390,438.096,-119.592,176.386,37.456,157.119
C02429=1067.381,437.852,-119.543,176.378,37.443,157.116
C02430=1067.373,437.606,-119.495,176.368,37.431,157.112
C02431=1067.363,437.361,-119.446,176.360,37.418,157.109
C02432=1067.354,437.116,-119.399,176.350,37.405,157.105
C02433=1067.345,436.870,-119.351,176.342,37.392,157.102
C02434=1067.335,436.626,-119.303,176.333,37.379,157.098
C02435=1067.326,436.380,-119.255,176.324,37.366,157.095
C02436=1067.317,436.134,-119.207,176.315,37.354,157.091
C02437=1067.308,435.889,-119.159,176.307,37.341,157.088
C02438=1067.299,435.644,-119.112,176.298,37.329,157.085
C02439=1067.290,435.400,-119.063,176.289,37.316,157.081
C02440=1067.281,435.155,-119.016,176.281,37.303,157.078
C02441=1067.271,434.909,-118.968,176.271,37.291,157.075
C02442=1067.263,434.664,-118.921,176.263,37.279,157.071
C02443=1067.253,434.419,-118.873,176.255,37.266,157.068
C02444=1067.245,434.173,-118.826,176.246,37.254,157.065
C02445=1067.236,433.928,-118.779,176.237,37.241,157.061
C02446=1067.227,433.682,-118.730,176.229,37.229,157.058
C02447=1067.218,433.437,-118.683,176.221,37.217,157.055
C02448=1067.210,433.192,-118.636,176.212,37.204,157.052
C02449=1067.201,432.947,-118.589,176.204,37.192,157.048
C02450=1067.191,432.701,-118.541,176.196,37.180,157.045
C02451=1067.183,432.456,-118.494,176.188,37.168,157.042
C02452=1067.174,432.211,-118.447,176.179,37.156,157.039
C02453=1067.165,431.966,-118.400,176.170,37.144,157.036
C02454=1067.156,431.721,-118.353,176.162,37.132,157.032
C02455=1067.148,431.475,-118.306,176.154,37.120,157.029
C02456=1067.139,431.230,-118.258,176.146,37.108,157.026
C02457=1067.130,430.984,-118.211,176.138,37.096,157.023
C02458=1067.121,430.739,-118.165,176.130,37.084,157.020
C02459=1067.112,430.493,-118.118,176.122,37.072,157.017
C02460=1067.104,430.248,-118.072,176.113,37.060,157.014
C02461=1067.095,430.003,-118.024,176.105,37.048,157.011
C02462=1067.086,429.757,-117.977,176.097,37.037,157.008
C02463=1067.078,429.512,-117.931,176.089,37.026,157.005
C02464=1067.068,429.267,-117.885,176.081,37.014,157.001
C02465=1067.060,429.021,-117.838,176.073,37.002,156.998
C02466=1067.049,428.708,-117.779,176.064,36.987,156.995
C02467=1067.038,428.394,-117.720,176.053,36.973,156.991
C02468=1067.027,428.082,-117.660,176.044,36.958,156.987
C02469=1067.016,427.768,-117.601,176.033,36.944,156.983
C02470=1067.008,427.522,-117.555,176.025,36.932,156.980
C02471=1066.999,427.277,-117.508,176.018,36.921,156.977
C02472=1066.990,427.031,-117.462,176.010,36.909,156.974
C02473=1066.981,426.785,-117.416,176.003,36.898,156.971
C02474=1066.973,426.541,-117.370,175.995,36.887,156.968
C02475=1066.965,426.295,-117.324,175.987,36.876,156.966
C02476=1066.955,426.050,-117.278,175.980,36.865,156.963
C02477=1066.947,425.803,-117.232,175.972,36.854,156.960
C02478=1066.938,425.558,-117.185,175.964,36.842,156.957
C02479=1066.930,425.313,-117.140,175.956,36.831,156.954
C02480=1066.922,425.067,-117.094,175.950,36.820,156.951
C02481=1066.913,424.821,-117.048,175.942,36.809,156.948
C02482=1066.904,424.575,-117.002,175.934,36.798,156.946
C02483=1066.896,424.330,-116.957,175.927,36.787,156.943
C02484=1066.887,424.084,-116.912,175.919,36.776,156.940
C02485=1066.879,423.838,-116.866,175.912,36.765,156.937
C02486=1066.870,423.593,-116.821,175.905,36.754,156.934
C02487=1066.862,423.347,-116.775,175.897,36.744,156.932
C02488=1066.854,423.102,-116.730,175.889,36.733,156.929
C02489=1066.845,422.856,-116.683,175.883,36.722,156.926
C02490=1066.837,422.611,-116.638,175.875,36.712,156.923
C02491=1066.829,422.364,-116.592,175.868,36.701,156.921
C02492=1066.820,422.119,-116.547,175.861,36.690,156.918
C02493=1066.812,421.873,-116.501,175.854,36.680,156.915
C02494=1066.803,421.627,-116.456,175.846,36.669,156.913
C02495=1066.795,421.382,-116.412,175.839,36.658,156.910
C02496=1066.788,421.136,-116.366,175.832,36.648,156.907
C02497=1066.779,420.890,-116.321,175.824,36.637,156.904
C02498=1066.771,420.645,-116.276,175.818,36.627,156.902
C02499=1066.762,420.398,-116.230,175.810,36.616,156.899
C02500=1066.754,420.153,-116.186,175.803,36.606,156.897
C02501=1066.745,419.907,-116.140,175.797,36.596,156.894
C02502=1066.737,419.661,-116.096,175.789,36.585,156.891
C02503=1066.728,419.415,-116.051,175.783,36.575,156.889
C02504=1066.721,419.169,-116.006,175.775,36.565,156.886
C02505=1066.713,418.924,-115.961,175.768,36.554,156.883
C02506=1066.704,418.678,-115.916,175.761,36.544,156.881
C02507=1066.696,418.432,-115.872,175.754,36.534,156.878
C02508=1066.688,418.186,-115.827,175.748,36.524,156.876
C02509=1066.679,417.940,-115.782,175.740,36.513,156.873
C02510=1066.671,417.695,-115.738,175.734,36.503,156.871
C02511=1066.663,417.449,-115.693,175.727,36.493,156.868
C02512=1066.655,417.203,-115.648,175.720,36.483,156.866
C02513=1066.647,416.956,-115.604,175.713,36.474,156.863
C02514=1066.638,416.711,-115.559,175.707,36.464,156.861
C02515=1066.630,416.465,-115.515,175.699,36.453,156.858
C02516=1066.622,416.219,-115.471,175.693,36.443,156.856
C02517=1066.614,415.973,-115.426,175.686,36.434,156.853
C02518=1066.606,415.728,-115.382,175.680,36.424,156.851
C02519=1066.598,415.481,-115.337,175.673,36.414,156.848
C02520=1066.589,415.235,-115.293,175.666,36.404,156.846
C02521=1066.582,414.989,-115.249,175.660,36.394,156.843
C02522=1066.573,414.696,-115.196,175.652,36.383,156.840
C02523=1066.563,414.402,-115.144,175.643,36.371,156.837
C02524=1066.553,414.109,-115.091,175.636,36.359,156.835
C02525=1066.543,413.815,-115.038,175.628,36.348,156.832
C02526=1066.536,413.569,-114.995,175.622,36.338,156.829
C02527=1066.528,413.323,-114.950,175.615,36.329,156.827
C02528=1066.519,413.077,-114.907,175.608,36.319,156.825
C02529=1066.511,412.831,-114.863,175.602,36.310,156.822
C02530=1066.503,412.585,-114.819,175.595,36.300,156.820
C02531=1066.495,412.339,-114.775,175.589,36.291,156.818
C02532=1066.487,412.093,-114.732,175.583,36.281,156.815
C02533=1066.479,411.847,-114.688,175.576,36.272,156.813
C02534=1066.471,411.601,-114.644,175.570,36.263,156.811
C02535=1066.463,411.354,-114.600,175.564,36.253,156.808
C02536=1066.455,411.108,-114.557,175.557,36.244,156.806
C02537=1066.447,410.863,-114.513,175.550,36.234,156.804
C02538=1066.439,410.616,-114.469,175.544,36.225,156.801
C02539=1066.431,410.371,-114.427,175.538,36.216,156.799
C02540=1066.423,410.125,-114.383,175.531,36.206,156.797
C02541=1066.415,409.878,-114.339,175.525,36.197,156.794
C02542=1066.408,409.632,-114.296,175.519,36.188,156.792
C02543=1066.399,409.386,-114.253,175.513,36.179,156.790
C02544=1066.392,409.140,-114.210,175.506,36.170,156.788
C02545=1066.384,408.894,-114.166,175.500,36.161,156.785
C02546=1066.376,408.648,-114.123,175.494,36.152,156.783
C02547=1066.368,408.401,-114.079,175.488,36.142,156.781
C02548=1066.361,408.156,-114.036,175.483,36.133,156.779
C02549=1066.352,407.910,-113.993,175.476,36.124,156.776
C02550=1066.345,407.663,-113.950,175.470,36.115,156.774
C02551=1066.338,407.417,-113.907,175.464,36.106,156.772
C02552=1066.329,407.171,-113.864,175.458,36.097,156.770
C02553=1066.322,406.925,-113.821,175.452,36.088,156.768
C02554=1066.314,406.678,-113.778,175.445,36.079,156.766
C02555=1066.306,406.432,-113.735,175.439,36.070,156.763
C02556=1066.299,406.187,-113.691,175.433,36.062,156.761
C02557=1066.291,405.940,-113.649,175.427,36.052,156.759
C02558=1066.283,405.694,-113.606,175.422,36.044,156.757
C02559=1066.275,405.448,-113.563,175.416,36.035,156.755
C02560=1066.268,405.201,-113.520,175.410,36.026,156.753
C02561=1066.260,404.955,-113.478,175.404,36.017,156.750
C02562=1066.252,404.709,-113.434,175.397,36.009,156.748
C02563=1066.245,404.463,-113.392,175.391,36.000,156.746
C02564=1066.236,404.216,-113.350,175.386,35.992,156.744
C02565=1066.229,403.970,-113.307,175.380,35.983,156.742
C02566=1066.221,403.724,-113.264,175.374,35.974,156.740
C02567=1066.214,403.478,-113.222,175.368,35.966,156.738
C02568=1066.206,403.232,-113.179,175.362,35.957,156.736
C02569=1066.198,402.985,-113.137,175.357,35.948,156.734
C02570=1066.191,402.739,-113.094,175.351,35.940,156.732
C02571=1066.183,402.493,-113.052,175.345,35.931,156.730
C02572=1066.175,402.247,-113.010,175.339,35.923,156.728
C02573=1066.168,402.001,-112.968,175.334,35.914,156.725
C02574=1066.160,401.754,-112.925,175.328,35.906,156.724
C02575=1066.153,401.508,-112.883,175.322,35.897,156.721
C02576=1066.145,401.261,-112.841,175.317,35.889,156.719
C02577=1066.137,401.015,-112.799,175.311,35.881,156.718
C02578=1066.128,400.726,-112.750,175.303,35.871,156.715
C02579=1066.119,400.436,-112.700,175.297,35.861,156.713
C02580=1066.111,400.147,-112.650,175.290,35.852,156.711
C02581=1066.102,399.858,-112.601,175.284,35.842,156.708
C02582=1066.094,399.611,-112.559,175.278,35.833,156.706
C02583=1066.086,399.365,-112.517,175.273,35.825,156.704
C02584=1066.079,399.119,-112.475,175.267,35.817,156.702
C02585=1066.071,398.873,-112.433,175.261,35.809,156.700
C02586=1066.063,398.626,-112.392,175.256,35.801,156.698
C02587=1066.056,398.380,-112.349,175.250,35.792,156.696
C02588=1066.049,398.134,-112.307,175.244,35.784,156.694
C02589=1066.041,397.887,-112.266,175.239,35.776,156.692
C02590=1066.034,397.641,-112.224,175.233,35.768,156.690
C02591=1066.027,397.395,-112.183,175.228,35.760,156.689
C02592=1066.019,397.149,-112.141,175.222,35.752,156.687
C02593=1066.011,396.901,-112.099,175.216,35.744,156.685
C02594=1066.003,396.655,-112.057,175.212,35.736,156.683
C02595=1065.996,396.409,-112.016,175.206,35.728,156.681
C02596=1065.989,396.162,-111.975,175.201,35.720,156.679
C02597=1065.981,395.916,-111.934,175.195,35.712,156.677
C02598=1065.973,395.670,-111.892,175.190,35.704,156.675
C02599=1065.966,395.424,-111.850,175.184,35.696,156.674
C02600=1065.958,395.177,-111.809,175.179,35.688,156.672
C02601=1065.951,394.931,-111.768,175.173,35.681,156.670
C02602=1065.944,394.684,-111.727,175.167,35.673,156.668
C02603=1065.936,394.438,-111.685,175.162,35.665,156.666
C02604=1065.929,394.192,-111.644,175.157,35.657,156.664
C02605=1065.922,393.945,-111.602,175.152,35.649,156.662
C02606=1065.910,393.545,-111.536,175.143,35.637,156.659
C02607=1065.898,393.146,-111.469,175.134,35.624,156.656
C02608=1065.885,392.745,-111.403,175.126,35.612,156.653
C02609=1065.873,392.346,-111.336,175.117,35.599,156.651
C02610=1065.866,392.100,-111.295,175.111,35.592,156.649
C02611=1065.859,391.853,-111.254,175.107,35.584,156.647
C02612=1065.851,391.607,-111.213,175.101,35.576,156.645
C02613=1065.844,391.360,-111.172,175.096,35.569,156.643
C02614=1065.836,391.113,-111.132,175.091,35.561,156.642
C02615=1065.830,390.867,-111.091,175.085,35.554,156.640
C02616=1065.822,390.621,-111.050,175.081,35.546,156.638
C02617=1065.814,390.375,-111.009,175.075,35.539,156.636
C02618=1065.807,390.127,-110.969,175.070,35.531,156.635
C02619=1065.799,389.881,-110.928,175.064,35.524,156.633
C02620=1065.793,389.635,-110.887,175.059,35.516,156.631
C02621=1065.785,389.388,-110.847,175.055,35.509,156.629
C02622=1065.778,389.142,-110.806,175.049,35.502,156.628
C02623=1065.770,388.895,-110.765,175.044,35.494,156.626
C02624=1065.763,388.649,-110.725,175.038,35.487,156.624
C02625=1065.755,388.403,-110.685,175.034,35.480,156.623
C02626=1065.748,388.156,-110.645,175.029,35.472,156.621
C02627=1065.741,387.910,-110.604,175.023,35.465,156.619
C02628=1065.733,387.663,-110.564,175.018,35.458,156.618
C02629=1065.726,387.416,-110.523,175.014,35.450,156.616
C02630=1065.715,387.050,-110.463,175.006,35.439,156.613
C02631=1065.704,386.684,-110.404,174.999,35.429,156.611
C02632=1065.694,386.319,-110.344,174.990,35.418,156.608
C02633=1065.683,385.952,-110.285,174.983,35.407,156.606
C02634=1065.676,385.705,-110.244,174.979,35.400,156.604
C02635=1065.668,385.460,-110.204,174.973,35.393,156.603
C02636=1065.661,385.212,-110.163,174.968,35.386,156.601
C02637=1065.654,384.966,-110.124,174.964,35.379,156.599
C02638=1065.647,384.719,-110.084,174.958,35.372,156.598
C02639=1065.640,384.473,-110.044,174.953,35.365,156.596
C02640=1065.632,384.226,-110.004,174.948,35.357,156.594
C02641=1065.625,383.980,-109.963,174.944,35.350,156.593
C02642=1065.618,383.733,-109.923,174.938,35.344,156.591
C02643=1065.611,383.487,-109.883,174.933,35.336,156.590
C02644=1065.603,383.240,-109.843,174.929,35.329,156.588
C02645=1065.597,382.993,-109.803,174.924,35.323,156.586
C02646=1065.589,382.746,-109.764,174.918,35.315,156.585
C02647=1065.583,382.499,-109.724,174.914,35.308,156.583
C02648=1065.576,382.253,-109.684,174.909,35.301,156.581
C02649=1065.568,382.006,-109.644,174.904,35.294,156.580
C02650=1065.562,381.760,-109.604,174.900,35.288,156.578
C02651=1065.555,381.514,-109.565,174.894,35.280,156.577
C02652=1065.547,381.267,-109.525,174.889,35.274,156.575
C02653=1065.540,381.020,-109.486,174.885,35.266,156.573
C02654=1065.532,380.773,-109.446,174.880,35.260,156.572
C02655=1065.526,380.526,-109.406,174.876,35.253,156.570
C02656=1065.519,380.280,-109.367,174.870,35.246,156.569
C02657=1065.512,380.033,-109.327,174.865,35.239,156.567
C02658=1065.504,379.786,-109.288,174.861,35.232,156.566
C02659=1065.498,379.540,-109.249,174.856,35.226,156.564
C02660=1065.490,379.293,-109.209,174.851,35.219,156.563
C02661=1065.483,379.046,-109.170,174.846,35.212,156.561
C02662=1065.476,378.800,-109.130,174.841,35.206,156.560
C02663=1065.469,378.552,-109.091,174.837,35.199,156.558
C02664=1065.461,378.306,-109.052,174.832,35.192,156.557
C02665=1065.455,378.059,-109.013,174.827,35.186,156.555
C02666=1065.448,377.813,-108.973,174.823,35.179,156.554
C02667=1065.440,377.565,-108.934,174.818,35.172,156.552
C02668=1065.433,377.319,-108.895,174.814,35.166,156.551
C02669=1065.426,377.072,-108.856,174.808,35.159,156.549
C02670=1065.419,376.826,-108.817,174.803,35.153,156.548
C02671=1065.413,376.579,-108.778,174.799,35.146,156.546
C02672=1065.405,376.332,-108.738,174.794,35.139,156.545
C02673=1065.398,376.085,-108.699,174.790,35.133,156.543
C02674=1065.391,375.838,-108.660,174.785,35.126,156.542
C02675=1065.384,375.591,-108.622,174.781,35.120,156.540
C02676=1065.378,375.345,-108.583,174.776,35.113,156.539
C02677=1065.370,375.098,-108.543,174.771,35.106,156.537
C02678=1065.363,374.852,-108.505,174.767,35.100,156.536
C02679=1065.356,374.604,-108.466,174.762,35.093,156.534
C02680=1065.349,374.357,-108.427,174.758,35.087,156.533
C02681=1065.342,374.111,-108.388,174.753,35.081,156.531
C02682=1065.335,373.866,-108.350,174.749,35.074,156.530
C02683=1065.329,373.621,-108.311,174.744,35.068,156.528
C02684=1065.322,373.376,-108.272,174.740,35.061,156.527
C02685=1065.315,373.132,-108.234,174.735,35.055,156.526
C02686=1065.309,372.887,-108.196,174.730,35.049,156.524
C02687=1065.301,372.642,-108.157,174.726,35.042,156.523
C02688=1065.295,372.398,-108.119,174.721,35.036,156.521
C02689=1065.287,372.154,-108.082,174.717,35.029,156.520
C02690=1065.280,371.906,-108.042,174.712,35.023,156.518
C02691=1065.273,371.659,-108.004,174.708,35.017,156.517
C02692=1065.266,371.413,-107.965,174.703,35.011,156.516
C02693=1065.259,371.165,-107.927,174.699,35.005,156.514
C02694=1065.252,370.918,-107.888,174.694,34.999,156.513
C02695=1065.245,370.672,-107.850,174.690,34.992,156.512
C02696=1065.238,370.425,-107.811,174.685,34.986,156.510
C02697=1065.231,370.178,-107.774,174.681,34.979,156.509
C02698=1065.224,369.931,-107.735,174.676,34.973,156.507
C02699=1065.217,369.684,-107.697,174.672,34.967,156.506
C02700=1065.210,369.438,-107.659,174.667,34.961,156.505
C02701=1065.204,369.191,-107.620,174.663,34.955,156.503
C02702=1065.196,368.944,-107.583,174.658,34.948,156.502
C02703=1065.190,368.697,-107.544,174.654,34.942,156.500
C02704=1065.183,368.450,-107.506,174.649,34.937,156.499
C02705=1065.176,368.203,-107.467,174.645,34.930,156.498
C02706=1065.169,367.956,-107.429,174.640,34.924,156.496
C02707=1065.162,367.709,-107.392,174.636,34.918,156.495
C02708=1065.155,367.462,-107.353,174.631,34.912,156.494
C02709=1065.149,367.215,-107.315,174.627,34.906,156.492
C02710=1065.141,366.968,-107.277,174.622,34.900,156.491
C02711=1065.135,366.721,-107.239,174.618,34.894,156.490
C02712=1065.128,366.474,-107.201,174.614,34.887,156.488
C02713=1065.121,366.227,-107.162,174.610,34.881,156.487
C02714=1065.114,365.981,-107.125,174.606,34.876,156.486
C02715=1065.108,365.733,-107.087,174.601,34.869,156.484
C02716=1065.101,365.486,-107.050,174.597,34.863,156.483
C02717=1065.094,365.239,-107.011,174.592,34.857,156.482
C02718=1065.087,364.992,-106.973,174.588,34.851,156.480
C02719=1065.081,364.745,-106.935,174.583,34.845,156.479
C02720=1065.074,364.498,-106.897,174.580,34.839,156.478
C02721=1065.067,364.251,-106.860,174.575,34.833,156.476
C02722=1065.060,364.004,-106.823,174.571,34.827,156.475
C02723=1065.054,363.757,-106.785,174.567,34.821,156.474
C02724=1065.046,363.510,-106.747,174.562,34.816,156.472
C02725=1065.039,363.263,-106.709,174.558,34.810,156.471
C02726=1065.033,363.016,-106.672,174.553,34.804,156.470
C02727=1065.026,362.769,-106.634,174.550,34.798,156.469
C02728=1065.019,362.522,-106.597,174.545,34.792,156.467
C02729=1065.013,362.275,-106.559,174.541,34.786,156.466
C02730=1065.006,362.028,-106.521,174.537,34.780,156.465
C02731=1064.998,361.781,-106.484,174.532,34.775,156.463
C02732=1064.991,361.533,-106.446,174.528,34.769,156.462
C02733=1064.985,361.287,-106.409,174.524,34.763,156.461
C02734=1064.978,361.039,-106.372,174.520,34.757,156.460
C02735=1064.972,360.793,-106.335,174.515,34.751,156.458
C02736=1064.964,360.545,-106.297,174.511,34.746,156.457
C02737=1064.957,360.298,-106.260,174.507,34.740,156.456
C02738=1064.951,360.062,-106.224,174.503,34.734,156.455
C02739=1064.945,359.827,-106.188,174.499,34.729,156.453
C02740=1064.938,359.591,-106.153,174.495,34.724,156.452
C02741=1064.932,359.354,-106.117,174.491,34.718,156.451
C02742=1064.925,359.119,-106.081,174.487,34.713,156.450
C02743=1064.919,358.882,-106.046,174.483,34.707,156.449
C02744=1064.913,358.647,-106.011,174.479,34.701,156.447
C02745=1064.906,358.411,-105.975,174.476,34.696,156.446
C02746=1064.900,358.163,-105.938,174.471,34.690,156.445
C02747=1064.893,357.917,-105.901,174.467,34.685,156.444
C02748=1064.886,357.669,-105.864,174.462,34.679,156.443
C02749=1064.880,357.423,-105.827,174.459,34.673,156.441
C02750=1064.873,357.175,-105.790,174.455,34.668,156.440
C02751=1064.866,356.928,-105.753,174.450,34.662,156.439
C02752=1064.859,356.681,-105.716,174.446,34.657,156.438
C02753=1064.853,356.434,-105.680,174.443,34.651,156.437
C02754=1064.845,356.186,-105.642,174.438,34.645,156.435
C02755=1064.839,355.939,-105.606,174.434,34.640,156.434
C02756=1064.832,355.692,-105.569,174.430,34.635,156.433
C02757=1064.826,355.445,-105.532,174.426,34.629,156.432
C02758=1064.819,355.197,-105.495,174.422,34.623,156.430
C02759=1064.812,354.950,-105.458,174.417,34.618,156.429
C02760=1064.805,354.703,-105.422,174.414,34.612,156.428
C02761=1064.799,354.456,-105.384,174.410,34.606,156.427
C02762=1064.792,354.208,-105.348,174.405,34.601,156.426
C02763=1064.785,353.961,-105.311,174.402,34.596,156.425
C02764=1064.779,353.714,-105.275,174.398,34.590,156.423
C02765=1064.772,353.467,-105.238,174.393,34.585,156.422
C02766=1064.765,353.220,-105.201,174.390,34.579,156.421
C02767=1064.758,352.973,-105.165,174.386,34.574,156.420
C02768=1064.751,352.726,-105.128,174.381,34.568,156.419
C02769=1064.745,352.479,-105.092,174.378,34.563,156.418
C02770=1064.739,352.232,-105.055,174.373,34.557,156.416
C02771=1064.732,351.984,-105.018,174.369,34.552,156.415
C02772=1064.726,351.737,-104.982,174.366,34.546,156.414
C02773=1064.719,351.490,-104.945,174.361,34.541,156.413
C02774=1064.712,351.242,-104.909,174.357,34.536,156.412
C02775=1064.705,350.995,-104.873,174.354,34.530,156.410
C02776=1064.699,350.748,-104.836,174.349,34.525,156.409
C02777=1064.692,350.500,-104.800,174.345,34.520,156.408
C02778=1064.685,350.253,-104.764,174.342,34.514,156.407
C02779=1064.679,350.006,-104.728,174.338,34.509,156.406
C02780=1064.672,349.758,-104.691,174.334,34.504,156.405
C02781=1064.666,349.511,-104.655,174.330,34.499,156.404
C02782=1064.658,349.264,-104.619,174.326,34.493,156.403
C02783=1064.652,349.017,-104.583,174.322,34.488,156.401
C02784=1064.645,348.769,-104.546,174.318,34.482,156.400
C02785=1064.638,348.522,-104.510,174.315,34.477,156.399
C02786=1064.632,348.274,-104.475,174.310,34.472,156.398
C02787=1064.626,348.027,-104.438,174.306,34.466,156.397
C02788=1064.618,347.780,-104.402,174.303,34.461,156.396
C02789=1064.612,347.532,-104.366,174.298,34.456,156.395
C02790=1064.606,347.285,-104.330,174.295,34.451,156.394
C02791=1064.599,347.039,-104.294,174.291,34.446,156.392
C02792=1064.593,346.791,-104.258,174.287,34.440,156.391
C02793=1064.587,346.544,-104.222,174.283,34.435,156.390
C02794=1064.580,346.310,-104.188,174.280,34.430,156.389
C02795=1064.574,346.076,-104.154,174.276,34.425,156.388
C02796=1064.568,345.842,-104.120,174.272,34.420,156.387
C02797=1064.561,345.608,-104.086,174.269,34.415,156.386
C02798=1064.555,345.374,-104.052,174.265,34.410,156.385
C02799=1064.549,345.140,-104.019,174.261,34.405,156.384
C02800=1064.543,344.906,-103.984,174.257,34.401,156.383
C02801=1064.537,344.673,-103.951,174.254,34.396,156.382
C02802=1064.530,344.424,-103.915,174.251,34.391,156.381
C02803=1064.523,344.178,-103.879,174.246,34.386,156.380
C02804=1064.517,343.930,-103.843,174.243,34.380,156.379
C02805=1064.510,343.683,-103.808,174.239,34.375,156.378
C02806=1064.504,343.435,-103.772,174.236,34.370,156.376
C02807=1064.497,343.188,-103.737,174.231,34.365,156.375
C02808=1064.491,342.940,-103.701,174.228,34.360,156.374
C02809=1064.484,342.694,-103.665,174.224,34.355,156.373
C02810=1064.477,342.446,-103.630,174.219,34.350,156.372
C02811=1064.471,342.199,-103.594,174.216,34.344,156.371
C02812=1064.464,341.951,-103.559,174.212,34.339,156.370
C02813=1064.458,341.704,-103.524,174.209,34.335,156.369
C02814=1064.452,341.456,-103.488,174.205,34.329,156.368
C02815=1064.444,341.209,-103.452,174.201,34.324,156.367
C02816=1064.438,340.962,-103.417,174.198,34.320,156.366
C02817=1064.432,340.714,-103.381,174.194,34.314,156.365
C02818=1064.425,340.467,-103.346,174.190,34.309,156.364
C02819=1064.418,340.220,-103.311,174.186,34.304,156.363
C02820=1064.412,339.972,-103.275,174.183,34.299,156.362
C02821=1064.405,339.725,-103.240,174.178,34.294,156.360
C02822=1064.399,339.477,-103.205,174.175,34.289,156.359
C02823=1064.393,339.230,-103.169,174.171,34.284,156.358
C02824=1064.386,338.982,-103.134,174.168,34.279,156.357
C02825=1064.379,338.735,-103.099,174.163,34.274,156.356
C02826=1064.373,338.487,-103.063,174.160,34.270,156.355
C02827=1064.366,338.240,-103.028,174.157,34.264,156.354
C02828=1064.360,337.992,-102.994,174.153,34.259,156.353
C02829=1064.353,337.745,-102.959,174.149,34.254,156.352
C02830=1064.348,337.498,-102.923,174.145,34.249,156.351
C02831=1064.341,337.250,-102.888,174.142,34.245,156.350
C02832=1064.334,337.003,-102.853,174.138,34.239,156.349
C02833=1064.328,336.755,-102.819,174.134,34.235,156.348
C02834=1064.321,336.507,-102.784,174.131,34.230,156.347
C02835=1064.314,336.260,-102.748,174.127,34.225,156.346
C02836=1064.307,336.013,-102.713,174.124,34.220,156.345
C02837=1064.302,335.764,-102.678,174.120,34.215,156.344
C02838=1064.295,335.517,-102.643,174.116,34.210,156.343
C02839=1064.289,335.270,-102.608,174.113,34.206,156.342
C02840=1064.282,335.022,-102.574,174.109,34.201,156.341
C02841=1064.275,334.775,-102.539,174.106,34.196,156.340
C02842=1064.269,334.528,-102.504,174.101,34.191,156.339
C02843=1064.262,334.280,-102.469,174.098,34.186,156.338
C02844=1064.256,334.033,-102.435,174.095,34.181,156.337
C02845=1064.250,333.785,-102.400,174.091,34.176,156.336
C02846=1064.243,333.538,-102.365,174.087,34.172,156.335
C02847=1064.236,333.290,-102.331,174.084,34.167,156.334
C02848=1064.230,333.042,-102.295,174.080,34.162,156.333
C02849=1064.224,332.795,-102.261,174.077,34.157,156.332
C02850=1064.217,332.559,-102.228,174.074,34.152,156.331
C02851=1064.212,332.323,-102.195,174.069,34.148,156.330
C02852=1064.205,332.086,-102.162,174.066,34.144,156.329
C02853=1064.199,331.850,-102.129,174.063,34.139,156.328
C02854=1064.193,331.614,-102.095,174.060,34.134,156.327
C02855=1064.187,331.377,-102.062,174.057,34.130,156.326
C02856=1064.180,331.141,-102.030,174.053,34.125,156.325
C02857=1064.175,330.904,-101.997,174.049,34.121,156.324
C02858=1064.168,330.657,-101.962,174.046,34.116,156.323
C02859=1064.162,330.410,-101.928,174.043,34.111,156.322
C02860=1064.155,330.162,-101.894,174.039,34.107,156.322
C02861=1064.148,329.914,-101.859,174.035,34.102,156.321
C02862=1064.142,329.666,-101.825,174.032,34.097,156.320
C02863=1064.135,329.420,-101.791,174.028,34.093,156.319
C02864=1064.128,329.172,-101.756,174.025,34.088,156.318
C02865=1064.122,328.924,-101.722,174.022,34.083,156.317
C02866=1064.115,328.677,-101.689,174.017,34.079,156.316
C02867=1064.109,328.429,-101.654,174.014,34.074,156.315
C02868=1064.102,328.181,-101.620,174.011,34.069,156.314
C02869=1064.095,327.933,-101.586,174.008,34.065,156.313
C02870=1064.089,327.686,-101.552,174.004,34.060,156.312
C02871=1064.082,327.438,-101.518,174.000,34.056,156.311
C02872=1064.076,327.191,-101.484,173.997,34.051,156.310
C02873=1064.070,326.943,-101.450,173.993,34.046,156.309
C02874=1064.063,326.695,-101.416,173.990,34.042,156.308
C02875=1064.057,326.448,-101.382,173.987,34.037,156.307
C02876=1064.050,326.200,-101.348,173.983,34.033,156.306
C02877=1064.043,325.952,-101.313,173.979,34.028,156.305
C02878=1064.037,325.705,-101.279,173.976,34.023,156.304
C02879=1064.030,325.457,-101.246,173.973,34.019,156.304
C02880=1064.024,325.210,-101.212,173.969,34.014,156.303
C02881=1064.017,324.962,-101.178,173.966,34.010,156.302
C02882=1064.011,324.715,-101.144,173.962,34.005,156.301
C02883=1064.005,324.467,-101.109,173.959,34.000,156.300
C02884=1063.998,324.220,-101.076,173.955,33.996,156.299
C02885=1063.992,323.972,-101.042,173.952,33.991,156.298
C02886=1063.985,323.725,-101.009,173.949,33.987,156.297
C02887=1063.979,323.477,-100.974,173.945,33.982,156.296
C02888=1063.972,323.230,-100.941,173.942,33.977,156.295
C02889=1063.966,322.981,-100.907,173.938,33.973,156.294
C02890=1063.960,322.734,-100.873,173.935,33.969,156.293
C02891=1063.953,322.486,-100.839,173.932,33.964,156.292
C02892=1063.947,322.239,-100.805,173.929,33.959,156.291
C02893=1063.940,321.991,-100.772,173.924,33.955,156.291
C02894=1063.934,321.743,-100.738,173.921,33.950,156.290
C02895=1063.928,321.496,-100.704,173.918,33.946,156.289
C02896=1063.922,321.248,-100.671,173.915,33.941,156.288
C02897=1063.915,321.001,-100.637,173.912,33.937,156.287
C02898=1063.909,320.753,-100.603,173.909,33.932,156.286
C02899=1063.902,320.505,-100.570,173.904,33.928,156.285
C02900=1063.897,320.258,-100.536,173.901,33.923,156.284
C02901=1063.890,320.010,-100.503,173.898,33.918,156.283
C02902=1063.884,319.762,-100.469,173.895,33.914,156.282
C02903=1063.877,319.515,-100.436,173.892,33.910,156.281
C02904=1063.871,319.267,-100.402,173.888,33.905,156.280
C02905=1063.865,319.019,-100.369,173.884,33.901,156.280
C02906=1063.859,318.780,-100.336,173.881,33.896,156.279
C02907=1063.853,318.540,-100.304,173.878,33.892,156.278
C02908=1063.847,318.302,-100.272,173.875,33.888,156.277
C02909=1063.840,318.063,-100.239,173.872,33.883,156.276
C02910=1063.835,317.823,-100.207,173.869,33.879,156.275
C02911=1063.829,317.584,-100.175,173.866,33.875,156.274
C02912=1063.823,317.345,-100.143,173.862,33.870,156.273
C02913=1063.817,317.105,-100.110,173.859,33.866,156.273
C02914=1063.810,316.858,-100.077,173.856,33.861,156.272
C02915=1063.804,316.611,-100.044,173.853,33.857,156.271
C02916=1063.798,316.363,-100.010,173.850,33.852,156.270
C02917=1063.791,316.115,-99.977,173.847,33.848,156.269
C02918=1063.786,315.867,-99.943,173.842,33.843,156.268
C02919=1063.779,315.619,-99.911,173.839,33.839,156.267
C02920=1063.774,315.372,-99.877,173.836,33.834,156.266
C02921=1063.767,315.125,-99.844,173.833,33.830,156.265
C02922=1063.761,314.877,-99.811,173.830,33.826,156.264
C02923=1063.755,314.628,-99.777,173.827,33.821,156.263
C02924=1063.748,314.381,-99.745,173.824,33.817,156.263
C02925=1063.743,314.133,-99.711,173.820,33.812,156.262
C02926=1063.736,313.886,-99.678,173.817,33.808,156.261
C02927=1063.730,313.638,-99.645,173.814,33.804,156.260
C02928=1063.723,313.390,-99.612,173.810,33.799,156.259
C02929=1063.717,313.142,-99.579,173.807,33.795,156.258
C02930=1063.710,312.895,-99.546,173.804,33.791,156.257
C02931=1063.704,312.647,-99.514,173.801,33.786,156.257
C02932=1063.697,312.399,-99.481,173.798,33.782,156.256
C02933=1063.691,312.151,-99.448,173.794,33.778,156.255
C02934=1063.685,311.904,-99.415,173.791,33.773,156.254
C02935=1063.678,311.656,-99.382,173.788,33.769,156.253
C02936=1063.672,311.409,-99.350,173.785,33.765,156.252
C02937=1063.664,311.161,-99.317,173.781,33.761,156.251
C02938=1063.658,310.912,-99.285,173.778,33.757,156.251
C02939=1063.652,310.665,-99.252,173.775,33.752,156.250
C02940=1063.646,310.417,-99.220,173.771,33.748,156.249
C02941=1063.640,310.170,-99.187,173.768,33.744,156.248
C02942=1063.633,309.922,-99.154,173.765,33.739,156.247
C02943=1063.626,309.674,-99.121,173.762,33.735,156.246
C02944=1063.620,309.426,-99.088,173.759,33.731,156.246
C02945=1063.614,309.178,-99.056,173.756,33.726,156.245
C02946=1063.607,308.931,-99.024,173.753,33.722,156.244
C02947=1063.601,308.683,-98.991,173.750,33.718,156.243
C02948=1063.595,308.435,-98.959,173.747,33.714,156.242
C02949=1063.589,308.187,-98.927,173.743,33.710,156.241
C02950=1063.582,307.940,-98.894,173.740,33.705,156.240
C02951=1063.576,307.692,-98.861,173.737,33.701,156.240
C02952=1063.570,307.444,-98.828,173.734,33.697,156.239
C02953=1063.564,307.196,-98.796,173.730,33.692,156.238
C02954=1063.557,306.949,-98.764,173.727,33.688,156.237
C02955=1063.550,306.701,-98.731,173.724,33.684,156.236
C02956=1063.544,306.453,-98.699,173.721,33.680,156.235
C02957=1063.538,306.206,-98.667,173.717,33.676,156.235
C02958=1063.532,305.957,-98.635,173.714,33.671,156.234
C02959=1063.526,305.710,-98.602,173.711,33.667,156.233
C02960=1063.519,305.462,-98.570,173.708,33.663,156.232
C02961=1063.513,305.214,-98.538,173.705,33.658,156.231
C02962=1063.507,304.977,-98.507,173.702,33.655,156.230
C02963=1063.501,304.739,-98.476,173.700,33.651,156.230
C02964=1063.495,304.502,-98.445,173.697,33.646,156.229
C02965=1063.489,304.264,-98.414,173.694,33.642,156.228
C02966=1063.483,304.027,-98.383,173.691,33.638,156.227
C02967=1063.477,303.790,-98.352,173.687,33.634,156.226
C02968=1063.471,303.553,-98.322,173.684,33.630,156.226
C02969=1063.465,303.315,-98.291,173.681,33.626,156.225
C02970=1063.459,303.068,-98.258,173.678,33.622,156.224
C02971=1063.453,302.820,-98.226,173.675,33.618,156.223
C02972=1063.447,302.572,-98.194,173.672,33.613,156.222
C02973=1063.440,302.325,-98.162,173.669,33.609,156.221
C02974=1063.434,302.076,-98.130,173.666,33.605,156.221
C02975=1063.428,301.829,-98.097,173.664,33.601,156.220
C02976=1063.422,301.581,-98.065,173.661,33.597,156.219
C02977=1063.416,301.333,-98.034,173.657,33.593,156.218
C02978=1063.409,301.086,-98.001,173.654,33.588,156.217
C02979=1063.403,300.838,-97.969,173.651,33.584,156.217
C02980=1063.397,300.589,-97.937,173.648,33.580,156.216
C02981=1063.391,300.342,-97.906,173.645,33.575,156.215
C02982=1063.385,300.095,-97.874,173.642,33.571,156.214
C02983=1063.379,299.846,-97.842,173.639,33.567,156.213
C02984=1063.373,299.598,-97.810,173.636,33.563,156.212
C02985=1063.366,299.350,-97.778,173.633,33.558,156.211
C02986=1063.361,299.103,-97.746,173.630,33.554,156.211
C02987=1063.355,298.855,-97.714,173.626,33.550,156.210
C02988=1063.349,298.607,-97.682,173.623,33.546,156.209
C02989=1063.342,298.359,-97.650,173.621,33.542,156.208
C02990=1063.336,298.112,-97.619,173.618,33.538,156.207
C02991=1063.330,297.863,-97.587,173.615,33.533,156.207
C02992=1063.324,297.615,-97.554,173.612,33.529,156.206
C02993=1063.318,297.368,-97.523,173.609,33.525,156.205
C02994=1063.312,297.120,-97.491,173.606,33.521,156.204
C02995=1063.306,296.872,-97.460,173.603,33.517,156.203
C02996=1063.300,296.624,-97.428,173.600,33.512,156.202
C02997=1063.294,296.376,-97.397,173.597,33.509,156.202
C02998=1063.288,296.128,-97.365,173.594,33.504,156.201
C02999=1063.281,295.880,-97.333,173.591,33.500,156.200
C03000=1063.275,295.632,-97.301,173.588,33.496,156.199
C03001=1063.269,295.385,-97.270,173.585,33.492,156.198
C03002=1063.263,295.137,-97.238,173.582,33.488,156.198
C03003=1063.256,294.889,-97.207,173.579,33.483,156.197
C03004=1063.249,294.641,-97.175,173.576,33.480,156.196
C03005=1063.244,294.393,-97.144,173.573,33.476,156.195
C03006=1063.237,294.145,-97.113,173.570,33.471,156.194
C03007=1063.231,293.897,-97.082,173.567,33.467,156.194
C03008=1063.225,293.649,-97.050,173.565,33.464,156.193
C03009=1063.219,293.402,-97.019,173.562,33.459,156.192
C03010=1063.212,293.154,-96.987,173.559,33.455,156.191
C03011=1063.207,292.906,-96.956,173.556,33.451,156.190
C03012=1063.200,292.658,-96.925,173.552,33.447,156.190
C03013=1063.193,292.410,-96.893,173.549,33.443,156.189
C03014=1063.188,292.162,-96.862,173.546,33.439,156.188
C03015=1063.182,291.914,-96.831,173.544,33.435,156.187
C03016=1063.175,291.666,-96.799,173.541,33.431,156.186
C03017=1063.169,291.419,-96.768,173.538,33.427,156.186
C03018=1063.163,291.188,-96.739,173.535,33.423,156.185
C03019=1063.157,290.959,-96.711,173.533,33.419,156.184
C03020=1063.152,290.728,-96.682,173.530,33.415,156.184
C03021=1063.145,290.499,-96.653,173.527,33.412,156.183
C03022=1063.140,290.269,-96.624,173.525,33.408,156.182
C03023=1063.134,290.039,-96.595,173.522,33.404,156.181
C03024=1063.129,289.810,-96.566,173.519,33.400,156.181
C03025=1063.123,289.580,-96.537,173.517,33.397,156.180
C03026=1063.117,289.332,-96.507,173.514,33.393,156.179
C03027=1063.110,289.084,-96.475,173.510,33.388,156.178
C03028=1063.105,288.836,-96.444,173.507,33.385,156.178
C03029=1063.098,288.588,-96.413,173.505,33.381,156.177
C03030=1063.092,288.340,-96.382,173.502,33.376,156.176
C03031=1063.086,288.093,-96.351,173.499,33.373,156.175
C03032=1063.079,287.844,-96.320,173.496,33.368,156.174
C03033=1063.073,287.596,-96.290,173.493,33.364,156.174
C03034=1063.067,287.348,-96.259,173.491,33.361,156.173
C03035=1063.061,287.101,-96.228,173.488,33.356,156.172
C03036=1063.054,286.853,-96.197,173.485,33.352,156.171
C03037=1063.048,286.604,-96.166,173.482,33.348,156.171
C03038=1063.042,286.356,-96.136,173.479,33.344,156.170
C03039=1063.035,286.108,-96.104,173.477,33.341,156.169
C03040=1063.029,285.861,-96.074,173.474,33.336,156.168
C03041=1063.023,285.612,-96.043,173.471,33.332,156.167
C03042=1063.017,285.364,-96.013,173.468,33.329,156.167
C03043=1063.010,285.116,-95.982,173.465,33.324,156.166
C03044=1063.005,284.868,-95.951,173.462,33.320,156.165
C03045=1062.998,284.620,-95.920,173.459,33.316,156.164
C03046=1062.992,284.372,-95.890,173.456,33.312,156.164
C03047=1062.986,284.124,-95.859,173.453,33.309,156.163
C03048=1062.980,283.876,-95.828,173.451,33.304,156.162
C03049=1062.974,283.629,-95.798,173.448,33.300,156.161
C03050=1062.968,283.380,-95.767,173.445,33.297,156.161
C03051=1062.962,283.132,-95.737,173.442,33.292,156.160
C03052=1062.955,282.884,-95.706,173.440,33.288,156.159
C03053=1062.949,282.637,-95.675,173.437,33.284,156.158
C03054=1062.943,282.388,-95.644,173.434,33.280,156.157
C03055=1062.937,282.140,-95.614,173.431,33.277,156.157
C03056=1062.931,281.892,-95.584,173.429,33.272,156.156
C03057=1062.925,281.644,-95.553,173.426,33.268,156.155
C03058=1062.919,281.396,-95.523,173.423,33.264,156.154
C03059=1062.913,281.147,-95.492,173.420,33.260,156.154
C03060=1062.907,280.900,-95.462,173.418,33.256,156.153
C03061=1062.901,280.652,-95.431,173.415,33.252,156.152
C03062=1062.895,280.403,-95.401,173.412,33.248,156.151
C03063=1062.888,280.156,-95.371,173.410,33.245,156.151
C03064=1062.882,279.908,-95.340,173.407,33.240,156.150
C03065=1062.876,279.659,-95.310,173.404,33.237,156.149
C03066=1062.870,279.412,-95.279,173.401,33.232,156.148
C03067=1062.863,279.163,-95.249,173.398,33.229,156.148
C03068=1062.857,278.916,-95.219,173.395,33.225,156.147
C03069=1062.851,278.668,-95.189,173.392,33.221,156.146
C03070=1062.845,278.419,-95.159,173.390,33.217,156.145
C03071=1062.838,278.171,-95.129,173.387,33.213,156.145
C03072=1062.833,277.923,-95.098,173.384,33.209,156.144
C03073=1062.826,277.675,-95.068,173.381,33.204,156.143
C03074=1062.821,277.450,-95.041,173.379,33.201,156.142
C03075=1062.815,277.226,-95.013,173.377,33.198,156.142
C03076=1062.810,277.001,-94.986,173.374,33.194,156.141
C03077=1062.804,276.777,-94.959,173.372,33.191,156.140
C03078=1062.799,276.553,-94.931,173.369,33.187,156.140
C03079=1062.793,276.328,-94.904,173.367,33.183,156.139
C03080=1062.788,276.104,-94.877,173.364,33.180,156.138
C03081=1062.782,275.880,-94.850,173.362,33.176,156.138
C03082=1062.775,275.631,-94.820,173.359,33.172,156.137
C03083=1062.770,275.383,-94.790,173.357,33.168,156.136
C03084=1062.764,275.135,-94.760,173.354,33.164,156.135
C03085=1062.757,274.888,-94.730,173.351,33.160,156.135
C03086=1062.751,274.638,-94.700,173.349,33.157,156.134
C03087=1062.745,274.391,-94.670,173.346,33.152,156.133
C03088=1062.739,274.143,-94.640,173.343,33.149,156.132
C03089=1062.733,273.895,-94.610,173.341,33.144,156.131
C03090=1062.726,273.646,-94.580,173.338,33.141,156.131
C03091=1062.721,273.398,-94.550,173.335,33.137,156.130
C03092=1062.714,273.150,-94.521,173.333,33.133,156.129
C03093=1062.709,272.902,-94.491,173.330,33.129,156.128
C03094=1062.702,272.654,-94.460,173.327,33.125,156.128
C03095=1062.696,272.405,-94.431,173.325,33.121,156.127
C03096=1062.690,272.158,-94.401,173.322,33.117,156.126
C03097=1062.684,271.909,-94.372,173.320,33.113,156.126
C03098=1062.677,271.661,-94.341,173.317,33.109,156.125
C03099=1062.671,271.413,-94.312,173.314,33.106,156.124
C03100=1062.665,271.165,-94.282,173.312,33.101,156.123
C03101=1062.659,270.917,-94.253,173.309,33.098,156.123
C03102=1062.652,270.669,-94.223,173.306,33.093,156.122
C03103=1062.647,270.421,-94.193,173.303,33.090,156.121
C03104=1062.640,270.172,-94.164,173.300,33.085,156.120
C03105=1062.634,269.924,-94.134,173.298,33.082,156.120
C03106=1062.628,269.676,-94.104,173.295,33.078,156.119
C03107=1062.623,269.428,-94.075,173.292,33.074,156.118
C03108=1062.616,269.180,-94.045,173.290,33.070,156.117
C03109=1062.610,268.932,-94.016,173.287,33.066,156.117
C03110=1062.604,268.683,-93.986,173.285,33.062,156.116
C03111=1062.597,268.435,-93.956,173.282,33.058,156.115
C03112=1062.591,268.187,-93.927,173.279,33.054,156.114
C03113=1062.585,267.939,-93.898,173.277,33.051,156.114
C03114=1062.579,267.691,-93.869,173.274,33.047,156.113
C03115=1062.573,267.443,-93.840,173.271,33.043,156.112
C03116=1062.567,267.195,-93.809,173.269,33.039,156.111
C03117=1062.560,266.946,-93.780,173.266,33.035,156.111
C03118=1062.554,266.698,-93.751,173.264,33.031,156.110
C03119=1062.548,266.449,-93.721,173.261,33.027,156.109
C03120=1062.542,266.201,-93.692,173.259,33.023,156.109
C03121=1062.536,265.954,-93.662,173.256,33.019,156.108
C03122=1062.529,265.706,-93.633,173.253,33.015,156.107
C03123=1062.524,265.457,-93.604,173.251,33.012,156.106
C03124=1062.518,265.209,-93.575,173.248,33.008,156.106
C03125=1062.511,264.961,-93.546,173.246,33.004,156.105
C03126=1062.506,264.712,-93.516,173.243,33.000,156.104
C03127=1062.500,264.464,-93.487,173.241,32.996,156.103
C03128=1062.493,264.216,-93.458,173.238,32.992,156.103
C03129=1062.487,263.968,-93.429,173.235,32.988,156.102
C03130=1062.481,263.745,-93.402,173.233,32.984,156.101
C03131=1062.476,263.523,-93.376,173.231,32.981,156.101
C03132=1062.471,263.300,-93.350,173.229,32.978,156.100
C03133=1062.465,263.077,-93.324,173.226,32.974,156.099
C03134=1062.459,262.855,-93.298,173.224,32.971,156.099
C03135=1062.454,262.632,-93.272,173.222,32.967,156.098
C03136=1062.448,262.409,-93.246,173.219,32.964,156.097
C03137=1062.443,262.187,-93.219,173.217,32.961,156.097
C03138=1062.436,261.939,-93.190,173.215,32.957,156.096
C03139=1062.430,261.690,-93.162,173.212,32.953,156.095
C03140=1062.423,261.442,-93.134,173.209,32.949,156.095
C03141=1062.417,261.194,-93.105,173.207,32.945,156.094
C03142=1062.411,260.946,-93.075,173.204,32.941,156.093
C03143=1062.405,260.698,-93.046,173.202,32.937,156.092
C03144=1062.398,260.450,-93.017,173.199,32.934,156.092
C03145=1062.392,260.200,-92.989,173.197,32.930,156.091
C03146=1062.386,259.952,-92.960,173.194,32.926,156.090
C03147=1062.379,259.704,-92.931,173.192,32.922,156.089
C03148=1062.373,259.456,-92.902,173.189,32.918,156.089
C03149=1062.367,259.207,-92.873,173.187,32.914,156.088
C03150=1062.361,258.959,-92.844,173.184,32.910,156.087
C03151=1062.355,258.711,-92.815,173.182,32.907,156.087
C03152=1062.349,258.463,-92.787,173.179,32.903,156.086
C03153=1062.342,258.215,-92.759,173.177,32.899,156.085
C03154=1062.336,257.967,-92.730,173.174,32.895,156.084
C03155=1062.330,257.719,-92.701,173.172,32.892,156.084
C03156=1062.324,257.470,-92.672,173.169,32.887,156.083
C03157=1062.318,257.222,-92.643,173.167,32.884,156.082
C03158=1062.312,256.973,-92.615,173.164,32.880,156.082
C03159=1062.305,256.725,-92.586,173.162,32.876,156.081
C03160=1062.299,256.477,-92.557,173.159,32.872,156.080
C03161=1062.293,256.228,-92.529,173.157,32.868,156.079
C03162=1062.286,255.980,-92.500,173.154,32.864,156.079
C03163=1062.280,255.732,-92.472,173.152,32.860,156.078
C03164=1062.274,255.483,-92.443,173.149,32.857,156.077
C03165=1062.269,255.235,-92.415,173.147,32.852,156.076
C03166=1062.262,254.987,-92.386,173.144,32.849,156.076
C03167=1062.257,254.739,-92.357,173.142,32.845,156.075
C03168=1062.250,254.490,-92.328,173.139,32.841,156.074
C03169=1062.244,254.242,-92.301,173.137,32.837,156.074
C03170=1062.237,253.994,-92.272,173.134,32.833,156.073
C03171=1062.231,253.745,-92.243,173.133,32.829,156.072
C03172=1062.226,253.498,-92.215,173.131,32.826,156.071
C03173=1062.220,253.249,-92.186,173.128,32.822,156.071
C03174=1062.214,253.001,-92.157,173.126,32.818,156.070
C03175=1062.208,252.752,-92.129,173.123,32.814,156.069
C03176=1062.201,252.504,-92.101,173.121,32.810,156.068
C03177=1062.195,252.255,-92.072,173.118,32.806,156.068
C03178=1062.189,252.007,-92.044,173.116,32.802,156.067
C03179=1062.183,251.759,-92.015,173.113,32.798,156.066
C03180=1062.177,251.511,-91.987,173.111,32.794,156.066
C03181=1062.170,251.262,-91.959,173.109,32.790,156.065
C03182=1062.165,251.015,-91.930,173.106,32.786,156.064
C03183=1062.159,250.766,-91.902,173.104,32.783,156.063
C03184=1062.153,250.517,-91.874,173.101,32.778,156.063
C03185=1062.147,250.268,-91.846,173.099,32.775,156.062
C03186=1062.141,250.046,-91.820,173.097,32.771,156.061
C03187=1062.136,249.822,-91.794,173.095,32.767,156.060
C03188=1062.131,249.598,-91.769,173.092,32.764,156.060
C03189=1062.125,249.374,-91.743,173.090,32.761,156.059
C03190=1062.121,249.151,-91.718,173.088,32.757,156.059
C03191=1062.114,248.928,-91.693,173.086,32.753,156.058
C03192=1062.109,248.703,-91.667,173.084,32.750,156.057
C03193=1062.104,248.480,-91.641,173.082,32.747,156.057
C03194=1062.098,248.232,-91.613,173.079,32.742,156.056
C03195=1062.091,247.983,-91.586,173.077,32.739,156.055
C03196=1062.086,247.734,-91.557,173.074,32.734,156.054
C03197=1062.080,247.486,-91.529,173.072,32.731,156.054
C03198=1062.074,247.238,-91.501,173.070,32.727,156.053
C03199=1062.067,246.990,-91.473,173.067,32.723,156.052
C03200=1062.062,246.742,-91.445,173.065,32.719,156.051
C03201=1062.056,246.493,-91.416,173.063,32.715,156.051
C03202=1062.050,246.244,-91.388,173.060,32.711,156.050
C03203=1062.044,245.997,-91.361,173.058,32.707,156.049
C03204=1062.038,245.748,-91.332,173.055,32.703,156.049
C03205=1062.031,245.499,-91.305,173.053,32.699,156.048
C03206=1062.026,245.251,-91.277,173.051,32.695,156.047
C03207=1062.019,245.003,-91.249,173.048,32.692,156.046
C03208=1062.013,244.754,-91.221,173.046,32.687,156.046
C03209=1062.007,244.506,-91.193,173.044,32.684,156.045
C03210=1062.001,244.258,-91.165,173.042,32.680,156.044
C03211=1061.995,244.009,-91.137,173.040,32.676,156.043
C03212=1061.989,243.761,-91.109,173.037,32.672,156.043
C03213=1061.983,243.512,-91.081,173.035,32.668,156.042
C03214=1061.977,243.263,-91.054,173.033,32.664,156.041
C03215=1061.972,243.015,-91.026,173.030,32.660,156.041
C03216=1061.965,242.767,-90.998,173.028,32.656,156.040
C03217=1061.960,242.519,-90.970,173.026,32.652,156.039
C03218=1061.953,242.270,-90.943,173.023,32.648,156.038
C03219=1061.946,242.022,-90.915,173.021,32.644,156.038
C03220=1061.941,241.774,-90.887,173.019,32.641,156.037
C03221=1061.935,241.525,-90.860,173.016,32.637,156.036
C03222=1061.928,241.276,-90.832,173.014,32.633,156.035
C03223=1061.923,241.028,-90.804,173.012,32.629,156.035
C03224=1061.916,240.780,-90.776,173.009,32.625,156.034
C03225=1061.910,240.531,-90.750,173.007,32.621,156.033
C03226=1061.904,240.283,-90.721,173.005,32.617,156.033
C03227=1061.897,240.034,-90.694,173.002,32.614,156.032
C03228=1061.892,239.786,-90.667,173.000,32.609,156.031
C03229=1061.886,239.537,-90.639,172.998,32.606,156.030
C03230=1061.880,239.289,-90.611,172.995,32.602,156.030
C03231=1061.873,239.041,-90.584,172.993,32.598,156.029
C03232=1061.867,238.793,-90.557,172.991,32.594,156.028
C03233=1061.861,238.544,-90.529,172.989,32.590,156.028
C03234=1061.855,238.295,-90.502,172.987,32.586,156.027
C03235=1061.849,238.047,-90.474,172.985,32.582,156.026
C03236=1061.842,237.799,-90.447,172.982,32.579,156.025
C03237=1061.836,237.550,-90.420,172.980,32.574,156.025
C03238=1061.830,237.301,-90.392,172.978,32.571,156.024
C03239=1061.825,237.053,-90.365,172.975,32.566,156.023
C03240=1061.818,236.805,-90.337,172.973,32.563,156.022
C03241=1061.812,236.557,-90.310,172.971,32.559,156.022
C03242=1061.807,236.330,-90.285,172.969,32.555,156.021
C03243=1061.801,236.103,-90.260,172.967,32.552,156.020
C03244=1061.795,235.876,-90.235,172.965,32.548,156.020
C03245=1061.790,235.649,-90.210,172.963,32.544,156.019
C03246=1061.784,235.422,-90.185,172.960,32.541,156.018
C03247=1061.779,235.196,-90.161,172.958,32.538,156.018
C03248=1061.774,234.969,-90.135,172.956,32.534,156.017
C03249=1061.768,234.742,-90.111,172.954,32.530,156.016
C03250=1061.761,234.494,-90.083,172.952,32.527,156.016
C03251=1061.756,234.245,-90.057,172.950,32.522,156.015
C03252=1061.749,233.998,-90.029,172.948,32.519,156.014
C03253=1061.744,233.748,-90.002,172.946,32.514,156.013
C03254=1061.738,233.500,-89.974,172.944,32.511,156.013
C03255=1061.731,233.251,-89.947,172.942,32.507,156.012
C03256=1061.726,233.003,-89.921,172.939,32.503,156.011
C03257=1061.719,232.755,-89.893,172.937,32.499,156.011
C03258=1061.713,232.506,-89.866,172.935,32.495,156.010
C03259=1061.707,232.258,-89.839,172.933,32.491,156.009
C03260=1061.701,232.009,-89.812,172.930,32.487,156.008
C03261=1061.695,231.761,-89.785,172.928,32.483,156.008
C03262=1061.689,231.512,-89.758,172.926,32.479,156.007
C03263=1061.682,231.264,-89.731,172.924,32.475,156.006
C03264=1061.676,231.015,-89.704,172.921,32.471,156.006
C03265=1061.671,230.766,-89.676,172.919,32.468,156.005
C03266=1061.665,230.518,-89.650,172.917,32.463,156.004
C03267=1061.659,230.270,-89.622,172.915,32.460,156.003
C03268=1061.653,230.021,-89.595,172.913,32.455,156.003
C03269=1061.647,229.773,-89.569,172.911,32.452,156.002
C03270=1061.641,229.524,-89.542,172.909,32.448,156.001
C03271=1061.634,229.276,-89.516,172.907,32.444,156.000
C03272=1061.628,229.027,-89.489,172.904,32.440,156.000
C03273=1061.622,228.779,-89.461,172.902,32.436,155.999
C03274=1061.616,228.531,-89.435,172.900,32.432,155.998
C03275=1061.610,228.282,-89.408,172.898,32.428,155.998
C03276=1061.604,228.033,-89.381,172.896,32.424,155.997
C03277=1061.597,227.784,-89.354,172.893,32.420,155.996
C03278=1061.591,227.536,-89.328,172.891,32.417,155.995
C03279=1061.585,227.288,-89.301,172.889,32.412,155.995
C03280=1061.579,227.039,-89.274,172.887,32.409,155.994
C03281=1061.573,226.790,-89.248,172.884,32.405,155.993
C03282=1061.567,226.542,-89.221,172.882,32.401,155.992
C03283=1061.560,226.293,-89.195,172.881,32.397,155.992
C03284=1061.554,226.045,-89.168,172.879,32.393,155.991
C03285=1061.549,225.797,-89.141,172.877,32.389,155.990
C03286=1061.542,225.547,-89.114,172.874,32.385,155.990
C03287=1061.536,225.299,-89.088,172.872,32.381,155.989
C03288=1061.530,225.051,-89.062,172.870,32.377,155.988
C03289=1061.524,224.803,-89.035,172.868,32.373,155.987
C03290=1061.518,224.554,-89.008,172.866,32.369,155.987
C03291=1061.512,224.305,-88.981,172.864,32.365,155.986
C03292=1061.506,224.057,-88.955,172.861,32.361,155.985
C03293=1061.499,223.808,-88.928,172.859,32.358,155.985
C03294=1061.493,223.560,-88.902,172.857,32.353,155.984
C03295=1061.488,223.311,-88.875,172.855,32.350,155.983
C03296=1061.482,223.063,-88.848,172.854,32.346,155.982
C03297=1061.476,222.814,-88.823,172.851,32.342,155.982
C03298=1061.470,222.583,-88.797,172.849,32.338,155.981
C03299=1061.464,222.353,-88.773,172.847,32.334,155.980
C03300=1061.459,222.122,-88.749,172.845,32.331,155.980
C03301=1061.453,221.891,-88.723,172.843,32.327,155.979
C03302=1061.448,221.661,-88.700,172.841,32.323,155.978
C03303=1061.441,221.430,-88.675,172.839,32.319,155.977
C03304=1061.436,221.199,-88.650,172.837,32.315,155.977
C03305=1061.431,220.968,-88.626,172.835,32.312,155.976
C03306=1061.424,220.720,-88.600,172.833,32.308,155.975
C03307=1061.418,220.471,-88.573,172.831,32.304,155.975
C03308=1061.412,220.223,-88.546,172.830,32.300,155.974
C03309=1061.406,219.974,-88.521,172.828,32.296,155.973
C03310=1061.400,219.726,-88.494,172.826,32.292,155.972
C03311=1061.393,219.477,-88.468,172.824,32.288,155.972
C03312=1061.388,219.228,-88.442,172.821,32.285,155.971
C03313=1061.381,218.980,-88.416,172.819,32.280,155.970
C03314=1061.375,218.732,-88.389,172.817,32.277,155.970
C03315=1061.369,218.483,-88.364,172.815,32.272,155.969
C03316=1061.363,218.234,-88.337,172.813,32.269,155.968
C03317=1061.356,217.986,-88.311,172.811,32.264,155.967
C03318=1061.351,217.737,-88.285,172.809,32.261,155.967
C03319=1061.344,217.489,-88.259,172.807,32.256,155.966
C03320=1061.339,217.240,-88.233,172.805,32.253,155.965
C03321=1061.332,216.992,-88.207,172.803,32.249,155.965
C03322=1061.327,216.743,-88.180,172.801,32.245,155.964
C03323=1061.320,216.494,-88.155,172.799,32.241,155.963
C03324=1061.314,216.246,-88.128,172.797,32.237,155.962
C03325=1061.308,215.997,-88.103,172.795,32.233,155.962
C03326=1061.302,215.749,-88.076,172.793,32.229,155.961
C03327=1061.296,215.500,-88.051,172.790,32.225,155.960
C03328=1061.290,215.252,-88.024,172.788,32.221,155.959
C03329=1061.284,215.003,-87.999,172.786,32.217,155.959
C03330=1061.278,214.755,-87.972,172.785,32.213,155.958
C03331=1061.272,214.506,-87.947,172.783,32.208,155.957
C03332=1061.266,214.257,-87.920,172.781,32.205,155.956
C03333=1061.259,214.008,-87.894,172.779,32.200,155.956
C03334=1061.253,213.760,-87.868,172.777,32.197,155.955
C03335=1061.247,213.511,-87.842,172.775,32.192,155.954
C03336=1061.241,213.262,-87.817,172.773,32.189,155.953
C03337=1061.235,213.014,-87.790,172.771,32.184,155.953
C03338=1061.229,212.765,-87.765,172.768,32.181,155.952
C03339=1061.224,212.516,-87.739,172.766,32.176,155.951
C03340=1061.217,212.268,-87.713,172.765,32.172,155.950
C03341=1061.211,212.020,-87.688,172.763,32.168,155.950
C03342=1061.205,211.771,-87.662,172.761,32.164,155.949
C03343=1061.199,211.523,-87.636,172.759,32.160,155.948
C03344=1061.193,211.274,-87.610,172.757,32.156,155.947
C03345=1061.187,211.025,-87.584,172.755,32.152,155.947
C03346=1061.181,210.777,-87.558,172.753,32.148,155.946
C03347=1061.175,210.528,-87.533,172.751,32.144,155.945
C03348=1061.168,210.280,-87.508,172.749,32.140,155.945
C03349=1061.163,210.031,-87.482,172.748,32.136,155.944
C03350=1061.156,209.783,-87.456,172.746,32.132,155.943
C03351=1061.150,209.534,-87.430,172.743,32.128,155.942
C03352=1061.144,209.285,-87.405,172.741,32.124,155.942
C03353=1061.138,209.036,-87.379,172.739,32.120,155.941
C03354=1061.132,208.808,-87.355,172.737,32.116,155.940
C03355=1061.126,208.580,-87.332,172.736,32.113,155.939
C03356=1061.121,208.351,-87.309,172.734,32.109,155.939
C03357=1061.115,208.124,-87.285,172.732,32.105,155.938
C03358=1061.110,207.896,-87.262,172.731,32.101,155.937
C03359=1061.104,207.667,-87.238,172.729,32.098,155.937
C03360=1061.099,207.439,-87.215,172.727,32.094,155.936
C03361=1061.093,207.210,-87.192,172.725,32.090,155.935
C03362=1061.068,206.162,-87.087,172.549,32.006,155.927
C03363=1061.062,205.913,-87.063,172.546,32.003,155.926
C03364=1061.057,205.664,-87.038,172.544,32.000,155.926
C03365=1061.051,205.416,-87.013,172.541,31.997,155.925
C03366=1061.045,205.167,-86.989,172.539,31.994,155.925
C03367=1061.039,204.918,-86.964,172.537,31.991,155.924
C03368=1061.032,204.669,-86.939,172.534,31.988,155.924
C03369=1061.027,204.421,-86.915,172.533,31.984,155.923
C03370=1061.021,204.171,-86.891,172.530,31.981,155.922
C03371=1061.016,203.923,-86.866,172.528,31.978,155.922
C03372=1061.010,203.674,-86.841,172.526,31.975,155.921
C03373=1061.004,203.426,-86.817,172.523,31.972,155.921
C03374=1060.998,203.177,-86.793,172.521,31.968,155.920
C03375=1060.992,202.929,-86.768,172.518,31.965,155.920
C03376=1060.986,202.679,-86.743,172.516,31.962,155.919
C03377=1060.981,202.431,-86.719,172.514,31.959,155.919
C03378=1060.975,202.181,-86.694,172.512,31.956,155.918
C03379=1060.969,201.934,-86.670,172.510,31.953,155.918
C03380=1060.963,201.684,-86.645,172.508,31.950,155.917
C03381=1060.958,201.436,-86.621,172.505,31.946,155.917
C03382=1060.951,201.187,-86.597,172.503,31.944,155.916
C03383=1060.946,200.938,-86.573,172.500,31.941,155.916
C03384=1060.939,200.689,-86.549,172.498,31.937,155.915
C03385=1060.934,200.441,-86.524,172.496,31.934,155.915
C03386=1060.927,200.192,-86.500,172.494,31.932,155.914
C03387=1060.921,199.944,-86.475,172.492,31.928,155.914
C03388=1060.915,199.695,-86.451,172.490,31.925,155.913
C03389=1060.909,199.446,-86.427,172.487,31.923,155.913
C03390=1060.904,199.197,-86.402,172.485,31.919,155.912
C03391=1060.898,198.949,-86.379,172.483,31.916,155.912
C03392=1060.892,198.699,-86.354,172.480,31.913,155.911
C03393=1060.886,198.451,-86.330,172.478,31.910,155.911
C03394=1060.880,198.202,-86.306,172.476,31.907,155.910
C03395=1060.874,197.954,-86.282,172.474,31.904,155.910
C03396=1060.868,197.704,-86.258,172.472,31.901,155.909
C03397=1060.862,197.456,-86.234,172.470,31.898,155.909
C03398=1060.856,197.207,-86.209,172.467,31.895,155.908
C03399=1060.850,196.958,-86.186,172.465,31.892,155.907
C03400=1060.844,196.710,-86.161,172.463,31.889,155.907
C03401=1060.838,196.461,-86.137,172.460,31.886,155.907
C03402=1060.833,196.212,-86.114,172.458,31.883,155.906
C03403=1060.826,195.963,-86.090,172.457,31.880,155.906
C03404=1060.821,195.714,-86.066,172.454,31.877,155.905
C03405=1060.815,195.466,-86.042,172.452,31.874,155.904
C03406=1060.809,195.217,-86.017,172.450,31.871,155.904
C03407=1060.803,194.968,-85.994,172.447,31.868,155.904
C03408=1060.797,194.719,-85.969,172.445,31.864,155.903
C03409=1060.791,194.471,-85.945,172.443,31.862,155.903
C03410=1060.786,194.221,-85.922,172.440,31.859,155.902
C03411=1060.779,193.972,-85.898,172.439,31.855,155.901
C03412=1060.774,193.724,-85.873,172.437,31.853,155.901
C03413=1060.768,193.476,-85.850,172.434,31.849,155.901
C03414=1060.761,193.227,-85.826,172.432,31.846,155.900
C03415=1060.756,192.977,-85.802,172.430,31.844,155.900
C03416=1060.750,192.729,-85.779,172.428,31.841,155.899
C03417=1060.744,192.480,-85.754,172.425,31.837,155.898
C03418=1060.738,192.232,-85.730,172.423,31.835,155.898
C03419=1060.733,191.982,-85.707,172.422,31.831,155.897
C03420=1060.727,191.733,-85.683,172.420,31.828,155.897
C03421=1060.722,191.485,-85.658,172.417,31.826,155.897
C03422=1060.715,191.237,-85.635,172.415,31.822,155.896
C03423=1060.709,190.952,-85.608,172.412,31.819,155.895
C03424=1060.703,190.670,-85.580,172.410,31.815,155.895
C03425=1060.696,190.386,-85.554,172.407,31.812,155.894
C03426=1060.689,190.102,-85.526,172.406,31.809,155.894
C03427=1060.684,189.853,-85.503,172.403,31.806,155.893
C03428=1060.678,189.605,-85.479,172.401,31.802,155.893
C03429=1060.672,189.357,-85.456,172.399,31.800,155.892
C03430=1060.666,189.107,-85.432,172.397,31.797,155.892
C03431=1060.660,188.858,-85.408,172.394,31.793,155.891
C03432=1060.655,188.610,-85.384,172.392,31.791,155.891
C03433=1060.649,188.361,-85.361,172.390,31.788,155.890
C03434=1060.643,188.113,-85.337,172.389,31.784,155.890
C03435=1060.638,187.863,-85.313,172.386,31.782,155.889
C03436=1060.632,187.614,-85.290,172.384,31.778,155.889
C03437=1060.627,187.365,-85.266,172.382,31.776,155.888
C03438=1060.620,187.117,-85.242,172.380,31.773,155.888
C03439=1060.615,186.868,-85.219,172.377,31.769,155.887
C03440=1060.609,186.619,-85.195,172.375,31.767,155.887
C03441=1060.603,186.370,-85.172,172.373,31.764,155.886
C03442=1060.598,186.121,-85.148,172.372,31.760,155.886
C03443=1060.592,185.872,-85.125,172.370,31.758,155.885
C03444=1060.586,185.624,-85.101,172.367,31.754,155.885
C03445=1060.581,185.375,-85.077,172.365,31.751,155.884
C03446=1060.575,185.127,-85.054,172.363,31.749,155.884
C03447=1060.569,184.877,-85.030,172.361,31.745,155.883
C03448=1060.563,184.628,-85.006,172.359,31.742,155.883
C03449=1060.558,184.380,-84.983,172.357,31.740,155.882
C03450=1060.552,184.131,-84.960,172.355,31.737,155.882
C03451=1060.546,183.882,-84.937,172.353,31.734,155.881
C03452=1060.540,183.633,-84.913,172.351,31.731,155.881
C03453=1060.534,183.384,-84.890,172.348,31.728,155.880
C03454=1060.528,183.136,-84.867,172.346,31.725,155.880
C03455=1060.522,182.887,-84.844,172.344,31.723,155.879
C03456=1060.515,182.637,-84.821,172.342,31.719,155.879
C03457=1060.509,182.388,-84.798,172.341,31.717,155.878
C03458=1060.503,182.140,-84.774,172.338,31.714,155.878
C03459=1060.497,181.891,-84.751,172.336,31.711,155.878
C03460=1060.492,181.642,-84.729,172.334,31.708,155.877
C03461=1060.485,181.393,-84.705,172.332,31.706,155.877
C03462=1060.479,181.145,-84.682,172.329,31.702,155.876
C03463=1060.474,180.896,-84.659,172.327,31.700,155.876
C03464=1060.468,180.647,-84.636,172.325,31.697,155.875
C03465=1060.462,180.398,-84.613,172.324,31.694,155.875
C03466=1060.455,180.149,-84.589,172.322,31.691,155.874
C03467=1060.449,179.900,-84.566,172.319,31.689,155.874
C03468=1060.443,179.651,-84.543,172.317,31.685,155.873
C03469=1060.438,179.402,-84.520,172.315,31.683,155.873
C03470=1060.432,179.154,-84.498,172.313,31.680,155.873
C03471=1060.426,178.905,-84.475,172.311,31.677,155.872
C03472=1060.420,178.656,-84.452,172.310,31.674,155.872
C03473=1060.413,178.407,-84.428,172.307,31.672,155.871
C03474=1060.407,178.158,-84.405,172.305,31.669,155.871
C03475=1060.402,177.909,-84.382,172.303,31.666,155.870
C03476=1060.396,177.660,-84.359,172.301,31.663,155.870
C03477=1060.390,177.412,-84.336,172.299,31.660,155.869
C03478=1060.384,177.163,-84.313,172.296,31.657,155.869
C03479=1060.379,176.914,-84.291,172.295,31.655,155.868
C03480=1060.372,176.665,-84.268,172.293,31.652,155.868
C03481=1060.366,176.416,-84.245,172.291,31.649,155.867
C03482=1060.361,176.167,-84.222,172.289,31.646,155.867
C03483=1060.355,175.918,-84.199,172.287,31.643,155.866
C03484=1060.349,175.669,-84.176,172.285,31.641,155.866
C03485=1060.343,175.420,-84.153,172.282,31.638,155.866
C03486=1060.336,175.171,-84.131,172.280,31.635,155.865
C03487=1060.331,174.888,-84.104,172.279,31.631,155.865
C03488=1060.324,174.604,-84.078,172.276,31.628,155.864
C03489=1060.317,174.320,-84.052,172.274,31.625,155.864
C03490=1060.310,174.036,-84.027,172.271,31.622,155.863
C03491=1060.305,173.787,-84.004,172.269,31.619,155.863
C03492=1060.299,173.538,-83.981,172.267,31.616,155.862
C03493=1060.292,173.290,-83.958,172.266,31.614,155.862
C03494=1060.287,173.041,-83.936,172.264,31.610,155.861
C03495=1060.281,172.792,-83.913,172.262,31.608,155.861
C03496=1060.275,172.543,-83.890,172.260,31.605,155.860
C03497=1060.269,172.294,-83.867,172.258,31.602,155.860
C03498=1060.263,172.045,-83.845,172.255,31.599,155.859
C03499=1060.258,171.796,-83.822,172.253,31.597,155.859
C03500=1060.252,171.547,-83.799,172.252,31.593,155.858
C03501=1060.246,171.298,-83.776,172.250,31.591,155.858
C03502=1060.240,171.049,-83.753,172.248,31.588,155.857
C03503=1060.234,170.801,-83.731,172.246,31.585,155.857
C03504=1060.228,170.551,-83.709,172.244,31.582,155.857
C03505=1060.223,170.302,-83.686,172.242,31.579,155.856
C03506=1060.217,170.053,-83.663,172.240,31.577,155.856
C03507=1060.211,169.805,-83.641,172.238,31.574,155.855
C03508=1060.205,169.557,-83.618,172.236,31.571,155.855
C03509=1060.200,169.307,-83.596,172.234,31.568,155.854
C03510=1060.194,169.058,-83.573,172.232,31.565,155.854
C03511=1060.188,168.810,-83.550,172.230,31.562,155.853
C03512=1060.182,168.561,-83.527,172.228,31.560,155.853
C03513=1060.177,168.311,-83.505,172.226,31.557,155.852
C03514=1060.171,168.062,-83.482,172.225,31.554,155.852
C03515=1060.164,167.814,-83.460,172.223,31.551,155.852
C03516=1060.160,167.565,-83.438,172.221,31.549,155.851
C03517=1060.154,167.316,-83.415,172.219,31.545,155.851
C03518=1060.148,167.067,-83.392,172.216,31.543,155.850
C03519=1060.142,166.818,-83.370,172.214,31.540,155.850
C03520=1060.136,166.569,-83.348,172.212,31.537,155.849
C03521=1060.130,166.320,-83.325,172.211,31.534,155.849
C03522=1060.125,166.070,-83.302,172.209,31.532,155.848
C03523=1060.119,165.823,-83.280,172.207,31.528,155.848
C03524=1060.113,165.574,-83.257,172.205,31.526,155.847
C03525=1060.108,165.324,-83.235,172.203,31.523,155.847
C03526=1060.102,165.076,-83.213,172.201,31.520,155.846
C03527=1060.096,164.826,-83.191,172.199,31.517,155.846
C03528=1060.091,164.578,-83.168,172.198,31.515,155.846
C03529=1060.086,164.328,-83.146,172.196,31.511,155.845
C03530=1060.079,164.080,-83.123,172.194,31.509,155.845
C03531=1060.073,163.831,-83.101,172.192,31.506,155.844
C03532=1060.068,163.581,-83.078,172.190,31.503,155.844
C03533=1060.062,163.334,-83.056,172.188,31.500,155.843
C03534=1060.057,163.084,-83.034,172.186,31.498,155.843
C03535=1060.051,162.835,-83.011,172.184,31.494,155.842
C03536=1060.045,162.586,-82.989,172.182,31.492,155.842
C03537=1060.040,162.338,-82.967,172.180,31.489,155.841
C03538=1060.034,162.088,-82.945,172.178,31.486,155.841
C03539=1060.028,161.839,-82.922,172.176,31.483,155.840
C03540=1060.022,161.590,-82.900,172.174,31.480,155.840
C03541=1060.018,161.341,-82.878,172.173,31.477,155.840
C03542=1060.012,161.092,-82.855,172.171,31.475,155.839
C03543=1060.006,160.843,-82.834,172.169,31.472,155.839
C03544=1059.999,160.595,-82.811,172.167,31.469,155.838
C03545=1059.994,160.346,-82.789,172.165,31.466,155.838
C03546=1059.988,160.097,-82.768,172.163,31.464,155.837
C03547=1059.982,159.848,-82.745,172.161,31.461,155.837
C03548=1059.976,159.598,-82.723,172.160,31.458,155.836
C03549=1059.970,159.349,-82.702,172.158,31.456,155.836
C03550=1059.964,159.101,-82.680,172.156,31.453,155.836
C03551=1059.958,158.816,-82.655,172.154,31.450,155.835
C03552=1059.951,158.533,-82.629,172.151,31.447,155.835
C03553=1059.944,158.248,-82.604,172.149,31.443,155.834
C03554=1059.937,157.963,-82.579,172.148,31.440,155.833
C03555=1059.932,157.715,-82.557,172.146,31.438,155.833
C03556=1059.926,157.466,-82.535,172.144,31.435,155.833
C03557=1059.920,157.217,-82.513,172.142,31.432,155.832
C03558=1059.915,156.968,-82.492,172.140,31.430,155.832
C03559=1059.908,156.719,-82.469,172.138,31.427,155.831
C03560=1059.902,156.470,-82.448,172.136,31.424,155.831
C03561=1059.896,156.221,-82.426,172.135,31.421,155.830
C03562=1059.891,155.972,-82.404,172.133,31.419,155.830
C03563=1059.885,155.723,-82.382,172.131,31.416,155.830
C03564=1059.879,155.474,-82.360,172.129,31.413,155.829
C03565=1059.873,155.225,-82.338,172.127,31.411,155.829
C03566=1059.868,154.976,-82.317,172.125,31.407,155.828
C03567=1059.861,154.727,-82.295,172.123,31.405,155.828
C03568=1059.855,154.478,-82.273,172.122,31.402,155.827
C03569=1059.850,154.229,-82.252,172.120,31.400,155.827
C03570=1059.844,153.980,-82.230,172.118,31.397,155.827
C03571=1059.838,153.731,-82.207,172.116,31.394,155.826
C03572=1059.832,153.482,-82.186,172.114,31.392,155.826
C03573=1059.826,153.234,-82.165,172.112,31.389,155.825
C03574=1059.820,152.984,-82.143,172.111,31.386,155.825
C03575=1059.815,152.735,-82.121,172.109,31.384,155.824
C03576=1059.809,152.486,-82.099,172.107,31.381,155.824
C03577=1059.803,152.237,-82.078,172.105,31.378,155.823
C03578=1059.797,151.988,-82.056,172.103,31.375,155.823
C03579=1059.791,151.739,-82.035,172.101,31.373,155.823
C03580=1059.785,151.490,-82.013,172.099,31.370,155.822
C03581=1059.780,151.241,-81.991,172.098,31.367,155.822
C03582=1059.774,150.992,-81.970,172.096,31.365,155.821
C03583=1059.768,150.743,-81.948,172.094,31.362,155.821
C03584=1059.762,150.494,-81.927,172.092,31.359,155.820
C03585=1059.756,150.245,-81.905,172.090,31.356,155.820
C03586=1059.750,149.996,-81.884,172.088,31.354,155.820
C03587=1059.744,149.748,-81.862,172.087,31.351,155.819
C03588=1059.738,149.498,-81.841,172.085,31.348,155.819
C03589=1059.732,149.249,-81.819,172.083,31.346,155.818
C03590=1059.727,149.000,-81.797,172.081,31.343,155.818
C03591=1059.721,148.751,-81.776,172.079,31.340,155.817
C03592=1059.715,148.503,-81.754,172.077,31.338,155.817
C03593=1059.709,148.253,-81.733,172.075,31.335,155.817
C03594=1059.703,148.004,-81.712,172.074,31.332,155.816
C03595=1059.698,147.755,-81.690,172.072,31.329,155.816
C03596=1059.692,147.506,-81.669,172.070,31.327,155.815
C03597=1059.686,147.257,-81.648,172.068,31.324,155.815
C03598=1059.680,147.008,-81.626,172.066,31.321,155.814
C03599=1059.674,146.759,-81.604,172.064,31.319,155.814
C03600=1059.668,146.510,-81.584,172.063,31.316,155.814
C03601=1059.662,146.261,-81.563,172.061,31.313,155.813
C03602=1059.656,146.012,-81.541,172.059,31.311,155.813
C03603=1059.650,145.763,-81.520,172.057,31.308,155.812
C03604=1059.644,145.514,-81.498,172.055,31.305,155.812
C03605=1059.639,145.265,-81.478,172.053,31.303,155.812
C03606=1059.632,145.016,-81.456,172.053,31.300,155.811
C03607=1059.627,144.767,-81.435,172.051,31.298,155.811
C03608=1059.621,144.518,-81.413,172.049,31.295,155.810
C03609=1059.615,144.268,-81.392,172.047,31.292,155.810
C03610=1059.609,144.020,-81.371,172.045,31.290,155.809
C03611=1059.602,143.771,-81.350,172.043,31.287,155.809
C03612=1059.597,143.522,-81.329,172.041,31.285,155.809
